TYPE "UDT_RATPositioning"
VERSION : 0.1
   STRUCT
      Lower { ExternalAccessible := 'False'; ExternalVisible := 'False'; ExternalWritable := 'False'} : Struct   // Roller part
         StartPositionA { ExternalAccessible := 'False'; ExternalVisible := 'False'; ExternalWritable := 'False'} : Int;   // Start position detected by OB30
         StartPositionB { ExternalAccessible := 'False'; ExternalVisible := 'False'; ExternalWritable := 'False'} : Int;
         EndPosition { ExternalAccessible := 'False'; ExternalVisible := 'False'; ExternalWritable := 'False'} : Int;   // End position defined by RAT FB
         Start { ExternalAccessible := 'False'; ExternalVisible := 'False'; ExternalWritable := 'False'} : Bool;   // Start command set by RAT FB
         Done { ExternalAccessible := 'False'; ExternalVisible := 'False'; ExternalWritable := 'False'} : Bool;   // MCO finish positioning
         ResetPosition { ExternalAccessible := 'False'; ExternalVisible := 'False'; ExternalWritable := 'False'} : Bool;
         PositionRequired { ExternalAccessible := 'False'; ExternalVisible := 'False'; ExternalWritable := 'False'} : Bool;
      END_STRUCT;
      Upper { ExternalAccessible := 'False'; ExternalVisible := 'False'; ExternalWritable := 'False'} : Struct   // UBT part
         StartPositionC { ExternalAccessible := 'False'; ExternalVisible := 'False'; ExternalWritable := 'False'} : Int;   // Start position detected by OB30
         StartPositionD { ExternalAccessible := 'False'; ExternalVisible := 'False'; ExternalWritable := 'False'} : Int;
         EndPosition { ExternalAccessible := 'False'; ExternalVisible := 'False'; ExternalWritable := 'False'} : Int;   // End position defined by RAT FB
         Start { ExternalAccessible := 'False'; ExternalVisible := 'False'; ExternalWritable := 'False'} : Bool;   // Start command set by RAT FB
         Done { ExternalAccessible := 'False'; ExternalVisible := 'False'; ExternalWritable := 'False'} : Bool;   // MCO finish positioning
         ResetPosition { ExternalAccessible := 'False'; ExternalVisible := 'False'; ExternalWritable := 'False'} : Bool;
         PositionRequired { ExternalAccessible := 'False'; ExternalVisible := 'False'; ExternalWritable := 'False'} : Bool;
      END_STRUCT;
   END_STRUCT;

END_TYPE

TYPE "UDT_ValveInterface"
TITLE = UDT_ValveInterface
VERSION : 0.1
//UDT valve interface between modules
   STRUCT
      Open { ExternalAccessible := 'False'; ExternalVisible := 'False'; ExternalWritable := 'False'} : Bool;   // Interface command valve Open / Extend
      Close { ExternalAccessible := 'False'; ExternalVisible := 'False'; ExternalWritable := 'False'} : Bool;   // Interface command valve Close / Retract
      IsOpened { ExternalAccessible := 'False'; ExternalVisible := 'False'; ExternalWritable := 'False'} : Bool;   // Valve feedback opened / extended
      IsClosed { ExternalAccessible := 'False'; ExternalVisible := 'False'; ExternalWritable := 'False'} : Bool;   // Valve feedback closed / retracted
      Error { ExternalAccessible := 'False'; ExternalVisible := 'False'; ExternalWritable := 'False'} : Bool;   // Valve error
   END_STRUCT;

END_TYPE

FUNCTION "FC_Fifo" : Void
TITLE = FC_Fifo
{ S7_Optimized_Access := 'TRUE' }
AUTHOR : MHSE
FAMILY : GeneralSystemFunctions
VERSION : 3.0
// ATTRIBUTES
// AUTO_NUMBER = True
// BLOCK_NUMBER = 17
// END_ATTRIBUTES
//Function for controlling FIFO register.
   VAR_INPUT
      ic_Mode : Char;   // Mode selector: "W" - Write; "R" - Read; "C" - Clear (Reset) "S" - Status
   END_VAR

   VAR_OUTPUT
      qUDT_Status : "UDT_FifoStatus";   // FIFO status structure
      qx_Error : Bool;   // Collective error output
      qx_Warning : Bool;   // Collective warning output
   END_VAR

   VAR_IN_OUT
      iqv_Data : Variant;   // Data
      iqUDT_FifoHeader : "UDT_FifoHeader";   // FIFO header
      iqv_DataBuffer : Variant;   // FIFO data buffer
   END_VAR

   VAR_TEMP
      tUDT_Status : "UDT_FifoStatus";   // Status structure
      ti_MoveBLKErrorCode : Int;   // Move_BLK_Variant function return
      tx_HeaderValid : Bool;   // Header valid
   END_VAR


BEGIN
	(*
	----------------------------------------------------------------------------------------

	Version history:
	Date        | Version   | Author        | Remark
	----------------------------------------------------------------------------------------
	24/05/2019  | 0.1       | L.Klar        | first release MHS TIA 15.1
	14/06/2019  | 0.2       | A.Nowak       | Replacement of instruction if for direct write into variable - Region 3 , 4.1 , 4.2 , 4.3 , 4.4 , 8.1  , 8.2
	17/07/2019  | 0.3       | L.Klar        | Status handling changed
	24/07/2019  | 2.0       | L.Klar        | 2.0 MHS library release TIA 15.1
	23/08/2019  | 2.1       | K.Pokorski    | Comments corrected
	27/08/2019  | 2.2       | M.Kurpiers    | Comments adjusted
	27/09/2019  | 2.3       | K.Pokorski    | Variant input included
	01/10/2019  | 2.4       | A.Nowak       | Correct comments and rename regions
	12/11/2019  | 3.0       | P.Majka       | 3.0 MHS library release TIA 15.1
	21/02/2023  | 4.0       | F.Baten       | 4.0 Release TIA 17.5
	*)

	REGION 1 – Diagnostic bits initialization

	    // Clear FIFO statuses
	    #tUDT_Status.FifoFull := FALSE;
	    #tUDT_Status.FifoPreFull := FALSE;

	END_REGION

	REGION 2 – Array's information

	    // If buffer elements type is invalid, set the error
	    #tUDT_Status.InvalidDataType := NOT (TypeOf(#iqv_Data) = TypeOfElements(#iqv_DataBuffer));

	END_REGION

	REGION 3 – Mode validation

	    // Set the mode invalid if selected mode isn't one of the following: W- Write, R - Read, C - Clear, S - Status
	    #tUDT_Status.InvalidMode := #ic_Mode <> 'W'
	    AND #ic_Mode <> 'R'
	    AND #ic_Mode <> 'C'
	    AND #ic_Mode <> 'S';

	END_REGION

	REGION 4 – The header settings checking

	    // The correct mode has been selected and data type is valid
	    IF (NOT #tUDT_Status.InvalidMode
	        AND NOT #tUDT_Status.InvalidDataType)
	    THEN

	        REGION 4.1 – The number of maximum FIFO entries validation

	            // Write the number of array's elements to FIFO header
	            #iqUDT_FifoHeader.MaxNrOfEntries := "FC_GetNrOfArrayEl"(#iqv_DataBuffer);

	            // Set the invalid maximum number of entries error
	            #tUDT_Status.InvalidMaxNrOfEntries := #iqUDT_FifoHeader.MaxNrOfEntries <= 0;

	        END_REGION

	        REGION 4.2 – The number of total FIFO entries validation

	            // Set the invalid total number of entries error
	            #tUDT_Status.InvalidTotalEntriesStored := #iqUDT_FifoHeader.TotalEntriesStored < 0        // The total number of entries is lower than 0
	            OR #iqUDT_FifoHeader.TotalEntriesStored > #iqUDT_FifoHeader.MaxNrOfEntries;               // The total number of entries is greater than the maximum number of entries

	        END_REGION

	        REGION 4.3 – The number of the next entry to write

	            // Set the invalid next entry to write
	            #tUDT_Status.InvalidNextEntryToWrite := #iqUDT_FifoHeader.NextEntryToWrite < 0            // The number of next entry to write is lower than 0
	            OR #iqUDT_FifoHeader.NextEntryToWrite >= #iqUDT_FifoHeader.MaxNrOfEntries;                // The number of next entry to write is greater or equal to the maximum number of entries

	        END_REGION

	        REGION 4.4 – The number of the next entry to read

	            // Set the invalid next entry to read
	            #tUDT_Status.InvalidNextEntryToRead := #iqUDT_FifoHeader.NextEntryToRead < 0              // The number of next entry to read is lower than 0
	            OR #iqUDT_FifoHeader.NextEntryToRead >= #iqUDT_FifoHeader.MaxNrOfEntries;                 // The number of next entry to read is greater or equal to the maximum nr of entries

	        END_REGION

	        REGION 4.5 – FIFO header validation summary

	            // Create collective header error
	            #tx_HeaderValid := NOT #tUDT_Status.InvalidMaxNrOfEntries
	            AND NOT #tUDT_Status.InvalidTotalEntriesStored
	            AND NOT #tUDT_Status.InvalidNextEntryToWrite
	            AND NOT #tUDT_Status.InvalidNextEntryToRead;

	        END_REGION

	    END_IF;

	END_REGION

	REGION 5 – Writing the data into the FIFO buffer

	    IF (#ic_Mode = 'W'                                                                          // Write mode selected
	        AND #tx_HeaderValid                                                                     // FIFO header valid
	        AND NOT #tUDT_Status.InvalidDataType)                                                  // Buffer data type valid
	    THEN


	        IF (#iqUDT_FifoHeader.TotalEntriesStored < #iqUDT_FifoHeader.MaxNrOfEntries)          // Checking total number of stored entries
	        THEN

	            // Move input data to FIFO data buffer
	            #ti_MoveBLKErrorCode := MOVE_BLK_VARIANT(SRC := #iqv_Data,
	                                                     COUNT := 1,
	                                                     SRC_INDEX := 0,
	                                                     DEST_INDEX := #iqUDT_FifoHeader.NextEntryToWrite,
	                                                     DEST => #iqv_DataBuffer);

	            // Increment the number of the next entry to write
	            #iqUDT_FifoHeader.NextEntryToWrite += 1;

	            // Increment the total number of stored entries
	            #iqUDT_FifoHeader.TotalEntriesStored += 1;


	            IF (#iqUDT_FifoHeader.NextEntryToWrite >= #iqUDT_FifoHeader.MaxNrOfEntries)       // Check the number of the next entry to write
	            THEN

	                #iqUDT_FifoHeader.NextEntryToWrite := 0;

	            END_IF;

	        ELSE

	            #tUDT_Status.FifoFull := TRUE;

	        END_IF;

	    END_IF;

	END_REGION

	REGION 6 – Reading the data from the FIFO data buffer

	    IF (#ic_Mode = 'R'                                                                  // Read mode selected
	        AND #tx_HeaderValid                                                             // FIFO header valid
	        AND NOT #tUDT_Status.InvalidDataType)                                           // Buffer data type valid
	    THEN

	        IF (#iqUDT_FifoHeader.TotalEntriesStored > 0)                                   // Checking total number of stored entries
	        THEN

	            // Move the FIFO data to the data output
	            #ti_MoveBLKErrorCode := MOVE_BLK_VARIANT(SRC := #iqv_DataBuffer,
	                                                     COUNT := 1,
	                                                     SRC_INDEX := #iqUDT_FifoHeader.NextEntryToRead,
	                                                     DEST_INDEX := 0,
	                                                     DEST => #iqv_Data);

	            // Increment the number of the next entry to read
	            #iqUDT_FifoHeader.NextEntryToRead += 1;

	            // Decrement the total number of stored entries
	            #iqUDT_FifoHeader.TotalEntriesStored -= 1;

	            IF (#iqUDT_FifoHeader.NextEntryToRead >= #iqUDT_FifoHeader.MaxNrOfEntries)  // Check the number of the next entry to read
	            THEN

	                #iqUDT_FifoHeader.NextEntryToRead := 0;

	            END_IF;

	        END_IF;

	    END_IF;

	END_REGION

	REGION 7 – Clearing the FIFO header

	    IF (#ic_Mode = 'C'                      // Clear mode selected
	        AND #tx_HeaderValid)                // FIFO header valid
	    THEN

	        #iqUDT_FifoHeader.TotalEntriesStored := 0;
	        #iqUDT_FifoHeader.NextEntryToWrite := 0;
	        #iqUDT_FifoHeader.NextEntryToRead := 0;

	    END_IF;

	END_REGION

	REGION 8 – FIFO management status update

	    IF (#tx_HeaderValid)                   // The header is valid
	    THEN

	        REGION 8.1 – FIFO Empty

	            // Set the FIFO empty status bit
	            #iqUDT_FifoHeader.Status.Empty := #iqUDT_FifoHeader.TotalEntriesStored = 0;

	        END_REGION

	        REGION 8.2 – FIFO Full

	            // Set the FIFO full status bit
	            #iqUDT_FifoHeader.Status.Full := #iqUDT_FifoHeader.TotalEntriesStored = #iqUDT_FifoHeader.MaxNrOfEntries;

	        END_REGION

	        REGION 8.3 – FIFO Pre-full

	            IF (#iqUDT_FifoHeader.TotalEntriesStored >= 0.9 * #iqUDT_FifoHeader.MaxNrOfEntries)       // Checking if the number of total stored entries is greater or equal to 90% of the max number of entries
	            THEN

	                // Set the FIFO pre-full status
	                #iqUDT_FifoHeader.Status.Prefull := TRUE;
	                #tUDT_Status.FifoPreFull := TRUE;

	            ELSE

	                #iqUDT_FifoHeader.Status.Prefull := FALSE;

	            END_IF;

	        END_REGION

	    END_IF;

	END_REGION

	REGION 9 – Status

	    REGION 9.1 – Common status update

	        // Collective error output
	        #qx_Error := NOT #tx_HeaderValid
	        OR #tUDT_Status.InvalidMode
	        OR #tUDT_Status.FifoFull
	        OR #tUDT_Status.InvalidDataType;

	        // Collective warning output
	        #qx_Warning := #tUDT_Status.FifoPreFull;

	    END_REGION

	    REGION 9.2 – Status update

	        // Update the outer status structure with internal status structure
	        #qUDT_Status := #tUDT_Status;

	    END_REGION

	END_REGION
END_FUNCTION

TYPE "UDT_VfdNordPI"
TITLE = UDT_VfdNordPI
VERSION : 0.1
//User-defined structure of VFD Nord input telegram.
   STRUCT
      ZSW : Struct   // Status word
         SetpointReached { ExternalAccessible := 'False'; ExternalVisible := 'False'; ExternalWritable := 'False'} : Bool;   // 0 = Actual value does not corresponf to setpoint. 1 = Actual value matches the setpoint
         BusControlActive { ExternalAccessible := 'False'; ExternalVisible := 'False'; ExternalWritable := 'False'} : Bool;   // 0 = Control on local device active. 1 = The master has beed requestd to take over control
         "StartFunction481.9" { ExternalAccessible := 'False'; ExternalVisible := 'False'; ExternalWritable := 'False'} : Bool;   // 1 = Bus bit 10 of status word is set P481
         RotationRightIsOn { ExternalAccessible := 'False'; ExternalVisible := 'False'; ExternalWritable := 'False'} : Bool;   // 1 = The FI output voltage has a RH rotation field
         RotationLeftIsOn { ExternalAccessible := 'False'; ExternalVisible := 'False'; ExternalWritable := 'False'} : Bool;   // 1 = The FI output voltage has a LH rotation field
         "StartFunction481.10" { ExternalAccessible := 'False'; ExternalVisible := 'False'; ExternalWritable := 'False'} : Bool;   // 1 = Bus bit 13 of status word is set P481
         ParameterSetBit0ON { ExternalAccessible := 'False'; ExternalVisible := 'False'; ExternalWritable := 'False'} : Bool;   // Parameter set bit 0 status
         ParameterSetBit1ON { ExternalAccessible := 'False'; ExternalVisible := 'False'; ExternalWritable := 'False'} : Bool;   // Parameter set bit 0 status
         ReadyToStart { ExternalAccessible := 'False'; ExternalVisible := 'False'; ExternalWritable := 'False'} : Bool;   // 1 = Initialisation completed, charging relay switched on, output voltage disabled
         ReadyForOperation { ExternalAccessible := 'False'; ExternalVisible := 'False'; ExternalWritable := 'False'} : Bool;   // 0 = No switch-on command present or fault. 1 = The inverted can start with the command "Enable operation"
         OperationEnabled { ExternalAccessible := 'False'; ExternalVisible := 'False'; ExternalWritable := 'False'} : Bool;   // 1 = The output voltage is enabled; ramp of the frequency inverter up to the existing setpoint
         Fault : Bool := FALSE;   // 1 = Drive unit defective, not ready for operation
         VoltageEnabled { ExternalAccessible := 'False'; ExternalVisible := 'False'; ExternalWritable := 'False'} : Bool;   // 0 = "Disable voltage" command present
         EmergencyStop { ExternalAccessible := 'False'; ExternalVisible := 'False'; ExternalWritable := 'False'} : Bool;   // 0 = "Emergency stop" command present
         StartingDisabled { ExternalAccessible := 'False'; ExternalVisible := 'False'; ExternalWritable := 'False'} : Bool;   // 1 = With the command "Standby" the FI goes into status "Ready to switch on"
         WarningActive { ExternalAccessible := 'False'; ExternalVisible := 'False'; ExternalWritable := 'False'} : Bool;   // 1 = Drive operation continues, no acknowledgement necessary
      END_STRUCT;
      ActualSpeed : Int;   // Actual calculated speed [rpm]. [Range  -200% ..200%][100%=4000HEX/ 16384DEC = P202 nominal speed]
      FaultCode : Int;   // Actual fault code
   END_STRUCT;

END_TYPE

DATA_BLOCK "DB_GINDefault"
{ S7_Optimized_Access := 'TRUE' }
VERSION : 0.1
NON_RETAIN
   VAR
      GIN { ExternalAccessible := 'False'; ExternalVisible := 'False'; ExternalWritable := 'False'; S7_SetPoint := 'False'} : Array[1..20] of "UDT_GIN";   // GIN informations
   END_VAR


BEGIN

END_DATA_BLOCK

FUNCTION_BLOCK "FB_VfdNORDCommissioning"
TITLE = Block for parameterising NORD VFD
{ S7_Optimized_Access := 'TRUE' }
VERSION : 0.1
// ATTRIBUTES
// AUTO_NUMBER = True
// BLOCK_NUMBER = 234
// END_ATTRIBUTES
   VAR_INPUT
      ihw_HardwareID { ExternalAccessible := 'False'; ExternalVisible := 'False'; ExternalWritable := 'False'} : HW_IO := 0;   // Device hardware ID
      iudt_MotorData { ExternalAccessible := 'False'; ExternalVisible := 'False'; ExternalWritable := 'False'} : "UDT_MotorData";
      ir_ReferenceFrequency { ExternalAccessible := 'False'; ExternalVisible := 'False'; ExternalWritable := 'False'} : Real;
      ix_VFDReadyToRun { ExternalAccessible := 'False'; ExternalVisible := 'False'; ExternalWritable := 'False'} : Bool;   // Condition to start motor identyfication
   END_VAR

   VAR_OUTPUT
      qi_HWAdress { ExternalAccessible := 'False'; ExternalVisible := 'False'; ExternalWritable := 'False'} : Int;
      qx_Busy { ExternalAccessible := 'False'; ExternalVisible := 'False'; ExternalWritable := 'False'} : Bool;   // Parametrisation in progress
      qx_Done { ExternalAccessible := 'False'; ExternalVisible := 'False'; ExternalWritable := 'False'} : Bool;   // Parametrisation done
      qx_Error { ExternalAccessible := 'False'; ExternalVisible := 'False'; ExternalWritable := 'False'} : Bool;   // Parametrisation error
      qx_24VCommissioningDone { ExternalAccessible := 'False'; ExternalVisible := 'False'; ExternalWritable := 'False'} : Bool;   // 24V commissioning done succesfully
   END_VAR

   VAR_IN_OUT
      iqx_Enable { ExternalAccessible := 'False'; ExternalVisible := 'False'; ExternalWritable := 'False'} : Bool;   // Input enable signal
   END_VAR

   VAR
      sFB_ParaAcycRead { ExternalAccessible := 'False'; ExternalVisible := 'False'; ExternalWritable := 'False'; S7_SetPoint := 'False'} : "FB_VfdNORDParaAcycRead";
      sFB_ParaAcycWrite { ExternalAccessible := 'False'; ExternalVisible := 'False'; ExternalWritable := 'False'; S7_SetPoint := 'False'} : "FB_VfdNORDParaAcycWrite";
      sR_TRIG_Done {InstructionName := 'R_TRIG'; LibVersion := '1.0'; ExternalAccessible := 'False'; ExternalVisible := 'False'; ExternalWritable := 'False'; S7_SetPoint := 'False'} : R_TRIG;
      sR_TRIG_StartJob {InstructionName := 'R_TRIG'; LibVersion := '1.0'; ExternalAccessible := 'False'; ExternalVisible := 'False'; ExternalWritable := 'False'; S7_SetPoint := 'False'} : R_TRIG;   // Bit for start trigger for rising edge
      sF_TRIG_CancelJob {InstructionName := 'F_TRIG'; LibVersion := '1.0'; ExternalAccessible := 'False'; ExternalVisible := 'False'; ExternalWritable := 'False'; S7_SetPoint := 'False'} : F_TRIG;   // Bit for start trigger for falling edge
      sa_Parameter { ExternalAccessible := 'False'; ExternalVisible := 'False'; ExternalWritable := 'False'; S7_SetPoint := 'False'} : Array[0..60] of "UDT_VfdNordParameter";   // Data of parameters
      sa_Status { ExternalAccessible := 'False'; ExternalVisible := 'False'; ExternalWritable := 'False'} : Struct   // Parametrization status
         StepNrError { ExternalAccessible := 'False'; ExternalVisible := 'False'; ExternalWritable := 'False'} : Int;   // The number of the step in witch the error occurred
         ParameterNrError { ExternalAccessible := 'False'; ExternalVisible := 'False'; ExternalWritable := 'False'} : Int;   // The number of the parameter in witch the error occurred
         StepNr { ExternalAccessible := 'False'; ExternalVisible := 'False'; ExternalWritable := 'False'} : Int := 0;   // Current step number
         ResponseValueError { ExternalAccessible := 'False'; ExternalVisible := 'False'; ExternalWritable := 'False'} : Bool;   // Response value error
         WrongFormat { ExternalAccessible := 'False'; ExternalVisible := 'False'; ExternalWritable := 'False'} : Bool;   // Wrong parameter format
         TimeExceeded { ExternalAccessible := 'False'; ExternalVisible := 'False'; ExternalWritable := 'False'} : Bool;   // Time has been exceeded
         NeedAck { ExternalAccessible := 'False'; ExternalVisible := 'False'; ExternalWritable := 'False'} : Bool;   // Need acknowledge signal (to cintinue parametrization)
         StepDone { ExternalAccessible := 'False'; ExternalVisible := 'False'; ExternalWritable := 'False'} : Bool;   // Step done
      END_STRUCT;
      si_StepTime { ExternalAccessible := 'False'; ExternalVisible := 'False'; ExternalWritable := 'False'} : Int;
      si_StepMax { ExternalAccessible := 'False'; ExternalVisible := 'False'; ExternalWritable := 'False'} : Int := 0;   // Maximum step number
      sx_Start { ExternalAccessible := 'False'; ExternalVisible := 'False'; ExternalWritable := 'False'} : Bool;   // Signal to start of parameterization function SinaPara
      sx_Busy { ExternalAccessible := 'False'; ExternalVisible := 'False'; ExternalWritable := 'False'} : Bool;   // Parametrization in progress (busy)
      sx_Done { ExternalAccessible := 'False'; ExternalVisible := 'False'; ExternalWritable := 'False'} : Bool;   // Parametrization done
      sx_Error { ExternalAccessible := 'False'; ExternalVisible := 'False'; ExternalWritable := 'False'} : Bool;   // Main error signal
      sx_PreparedData { ExternalAccessible := 'False'; ExternalVisible := 'False'; ExternalWritable := 'False'} : Bool;   // Step data prepared
      sx_ReadOrder { ExternalAccessible := 'False'; ExternalVisible := 'False'; ExternalWritable := 'False'} : Bool;   // Order to read paraeter with transition from 0 to 1
      sx_WriteOrder { ExternalAccessible := 'False'; ExternalVisible := 'False'; ExternalWritable := 'False'} : Bool;   // Order to write parameter with transition from 0 to 1
      sx_MaxStepCalculation { ExternalAccessible := 'False'; ExternalVisible := 'False'; ExternalWritable := 'False'} : Bool;   // Maximum step calculated
   END_VAR
   VAR RETAIN
      sx_24VCommissioningDone { ExternalAccessible := 'False'; ExternalVisible := 'False'; ExternalWritable := 'False'} : Bool;   // 24V commissioning done succesfully
   END_VAR

   VAR_TEMP
      ti_index : Int;   // Temporary array index
      ti_ControlMethod : Int;
      ti_EncoderCode : Int;
      ti_i : Int;   // Loop counter
      ti_BrakeReaction : Int;
   END_VAR

   VAR CONSTANT
      ci_CFC_ClosedLoop : Int := 1;
      ci_CFC_OpenLoop : Int := 0;
      ci_EncoderRes512 : Int := 1;
      ci_EncoderRes1024 : Int := 3;
      ci_EncoderRes2048 : Int := 5;
      ci_EncoderRes4096 : Int := 6;
      ci_MaxStepTime : Int := 100;
   END_VAR


BEGIN
	(*
	----------------------------------------------------------------------------------------

	Version history:
	Date        | Version   | Author        | Remark
	----------------------------------------------------------------------------------------
	12/01/2020  | 0.1       | S.Theocharis  | Initial version TIA 15.1
	08/04/2021  | 0.2       | F.Baten       | New read/write blocks
	                                        | New motor parameter set ( most values not 32bit )
	                                        | PN device with onboard safety
	                                        | Reading and writing optimised
	27/01/2022  | 0.3       | K.Pokorski    | Add 24V and 400V commissionig status
	                                        | Fix VFD Output bug
	                                        | Initialize InUse status in all parameters
	                                        | Fix Motor identification
	                                        | Save parameters to External memory
	                                        | Delete saving F-parameters from sequence (not working and creating faults)
	                                        | Delete reading CRC code (reading old CRC code what can be confusing)
	21/04/2022  | 0.4       | K.Pokorski    | Delete motor identification
	21/02/2023  | 4.0       | F.Baten       | 4.0 Release TIA 17.5

	*)

	REGION 1 - Start Job

	    // Monitor rising trigger if is input enable signal
	    #sR_TRIG_StartJob(CLK := #iqx_Enable);

	    IF (#sR_TRIG_StartJob.Q)
	    THEN
	        #sx_Start := TRUE;
	        #sx_Busy := TRUE;
	        #sx_Done := FALSE;
	        #sx_Error := FALSE;
	        #sx_PreparedData := FALSE;
	        #sx_MaxStepCalculation := FALSE;
	        #sa_Status.StepDone := FALSE;
	        #sa_Status.StepNrError := 0;
	        #sa_Status.ParameterNrError := 0;
	        #sa_Status.StepNr := 0;
	        #si_StepTime := 0;
	        #qi_HWAdress := 0;

	        FOR #ti_i := 0 TO 60 DO
	            #sa_Parameter[#ti_i].InUse := FALSE;
	        END_FOR;



	    END_IF;

	END_REGION

	REGION 2 - Build Sequences in static memory

	    IF #sR_TRIG_StartJob.Q THEN
	        //  IF NOT #sx_24VCommissioningDone THEN
	        REGION Step 01 - P523 Factory reset [0..3]
	            #ti_index := 0;
	            #sa_Parameter[#ti_index].ParaNumber := 523;
	            #sa_Parameter[#ti_index].Index := 0;
	            #sa_Parameter[#ti_index].WriteValue := 1;
	            #sa_Parameter[#ti_index].WriteAccess := TRUE;
	            #sa_Parameter[#ti_index].ParaSet := 0;
	            #sa_Parameter[#ti_index].Format32 := FALSE;
	            #sa_Parameter[#ti_index].ActualValue := 0;
	            #sa_Parameter[#ti_index].InUse := TRUE;
	            #sa_Parameter[#ti_index].RamOnly := FALSE;
	        END_REGION

	        REGION Step 02 - P003 Set supervisor code to access all parameters [0..9999]
	            #ti_index := #ti_index + 1;
	            #sa_Parameter[#ti_index].ParaNumber := 3;
	            #sa_Parameter[#ti_index].Index := 0;
	            #sa_Parameter[#ti_index].WriteValue := 3;
	            #sa_Parameter[#ti_index].WriteAccess := TRUE;
	            #sa_Parameter[#ti_index].ParaSet := 0;
	            #sa_Parameter[#ti_index].Format32 := FALSE;
	            #sa_Parameter[#ti_index].ActualValue := 0;
	            #sa_Parameter[#ti_index].InUse := TRUE;
	            #sa_Parameter[#ti_index].RamOnly := FALSE;
	        END_REGION

	        REGION Step 03 - P800 Set Operating mode Safety [0-1]
	            #ti_index := #ti_index + 1;
	            #sa_Parameter[#ti_index].ParaNumber := 800;
	            #sa_Parameter[#ti_index].Index := 1;
	            #sa_Parameter[#ti_index].WriteValue := 1;
	            #sa_Parameter[#ti_index].WriteAccess := TRUE;
	            #sa_Parameter[#ti_index].ParaSet := 0;
	            #sa_Parameter[#ti_index].Format32 := FALSE;
	            #sa_Parameter[#ti_index].ActualValue := 0;
	            #sa_Parameter[#ti_index].InUse := TRUE;
	            #sa_Parameter[#ti_index].RamOnly := FALSE;
	        END_REGION

	        REGION Step 04 - P800 Set Operating mode Safety [0-1]
	            #ti_index := #ti_index + 1;
	            #sa_Parameter[#ti_index].ParaNumber := 800;
	            #sa_Parameter[#ti_index].Index := 2;
	            #sa_Parameter[#ti_index].WriteValue := 0;
	            #sa_Parameter[#ti_index].WriteAccess := TRUE;
	            #sa_Parameter[#ti_index].ParaSet := 0;
	            #sa_Parameter[#ti_index].Format32 := FALSE;
	            #sa_Parameter[#ti_index].ActualValue := 0;
	            #sa_Parameter[#ti_index].InUse := TRUE;
	            #sa_Parameter[#ti_index].RamOnly := FALSE;
	        END_REGION

	        REGION Step 05 - P802 Set Enable safety channel [0-1]  Channel 1 on
	            #ti_index := #ti_index + 1;
	            #sa_Parameter[#ti_index].ParaNumber := 802;
	            #sa_Parameter[#ti_index].Index := 1;
	            #sa_Parameter[#ti_index].WriteValue := 1;
	            #sa_Parameter[#ti_index].WriteAccess := TRUE;
	            #sa_Parameter[#ti_index].ParaSet := 0;
	            #sa_Parameter[#ti_index].Format32 := FALSE;
	            #sa_Parameter[#ti_index].ActualValue := 0;
	            #sa_Parameter[#ti_index].InUse := TRUE;
	            #sa_Parameter[#ti_index].RamOnly := FALSE;
	        END_REGION

	        REGION Step 06 - P802 Set Enable safety channel [0-1]  Channel 2 on
	            #ti_index := #ti_index + 1;
	            #sa_Parameter[#ti_index].ParaNumber := 802;
	            #sa_Parameter[#ti_index].Index := 2;
	            #sa_Parameter[#ti_index].WriteValue := 1;
	            #sa_Parameter[#ti_index].WriteAccess := TRUE;
	            #sa_Parameter[#ti_index].ParaSet := 0;
	            #sa_Parameter[#ti_index].Format32 := FALSE;
	            #sa_Parameter[#ti_index].ActualValue := 0;
	            #sa_Parameter[#ti_index].InUse := TRUE;
	            #sa_Parameter[#ti_index].RamOnly := FALSE;
	        END_REGION

	        REGION Step 07 - P802 Set Enable safety channel [0-1]  Channel 3 on
	            #ti_index := #ti_index + 1;
	            #sa_Parameter[#ti_index].ParaNumber := 802;
	            #sa_Parameter[#ti_index].Index := 3;
	            #sa_Parameter[#ti_index].WriteValue := 1;
	            #sa_Parameter[#ti_index].WriteAccess := TRUE;
	            #sa_Parameter[#ti_index].ParaSet := 0;
	            #sa_Parameter[#ti_index].Format32 := FALSE;
	            #sa_Parameter[#ti_index].ActualValue := 0;
	            #sa_Parameter[#ti_index].InUse := TRUE;
	            #sa_Parameter[#ti_index].RamOnly := FALSE;
	        END_REGION

	        REGION Step 08 - P846 Read dipswitches
	            #ti_index := #ti_index + 1;
	            #sa_Parameter[#ti_index].ParaNumber := 846;
	            #sa_Parameter[#ti_index].Index := 0;
	            #sa_Parameter[#ti_index].WriteValue := 0;
	            #sa_Parameter[#ti_index].WriteAccess := FALSE;
	            #sa_Parameter[#ti_index].ParaSet := 0;
	            #sa_Parameter[#ti_index].Format32 := FALSE;
	            #sa_Parameter[#ti_index].ActualValue := 0;
	            #sa_Parameter[#ti_index].InUse := TRUE;
	            #sa_Parameter[#ti_index].RamOnly := FALSE;
	        END_REGION

	        REGION Step 09 - P120 Set extern control units [0-1]  Switch off 3 and 4
	            #ti_index := #ti_index + 1;
	            #sa_Parameter[#ti_index].ParaNumber := 120;
	            #sa_Parameter[#ti_index].Index := 3;
	            #sa_Parameter[#ti_index].WriteValue := 0;
	            #sa_Parameter[#ti_index].WriteAccess := TRUE;
	            #sa_Parameter[#ti_index].ParaSet := 0;
	            #sa_Parameter[#ti_index].Format32 := FALSE;
	            #sa_Parameter[#ti_index].ActualValue := 0;
	            #sa_Parameter[#ti_index].InUse := TRUE;
	            #sa_Parameter[#ti_index].RamOnly := FALSE;
	        END_REGION

	        REGION Step 10 - P120 Set extern control units [0-1]  Switch off 3 and 4
	            #ti_index := #ti_index + 1;
	            #sa_Parameter[#ti_index].ParaNumber := 120;
	            #sa_Parameter[#ti_index].Index := 4;
	            #sa_Parameter[#ti_index].WriteValue := 0;
	            #sa_Parameter[#ti_index].WriteAccess := TRUE;
	            #sa_Parameter[#ti_index].ParaSet := 0;
	            #sa_Parameter[#ti_index].Format32 := FALSE;
	            #sa_Parameter[#ti_index].ActualValue := 0;
	            #sa_Parameter[#ti_index].InUse := TRUE;
	            #sa_Parameter[#ti_index].RamOnly := FALSE;
	        END_REGION

	        REGION Step 11 - P202 Write motor nominal speed [150...24000]rpm
	            #ti_index := #ti_index + 1;
	            #sa_Parameter[#ti_index].ParaNumber := 202;
	            #sa_Parameter[#ti_index].Index := 0;
	            #sa_Parameter[#ti_index].WriteValue := #iudt_MotorData.NominalSpeed;
	            #sa_Parameter[#ti_index].WriteAccess := TRUE;
	            #sa_Parameter[#ti_index].ParaSet := 1; // Parameter set 1
	            #sa_Parameter[#ti_index].Format32 := FALSE;
	            #sa_Parameter[#ti_index].ActualValue := 0;
	            #sa_Parameter[#ti_index].InUse := TRUE;
	            #sa_Parameter[#ti_index].RamOnly := FALSE;
	        END_REGION

	        REGION Step 12 - P203 Write motor nominal current [0.1 ...1000.0]A
	            #ti_index := #ti_index + 1;
	            #sa_Parameter[#ti_index].ParaNumber := 203;
	            #sa_Parameter[#ti_index].Index := 0;
	            #sa_Parameter[#ti_index].WriteValue := (REAL_TO_DINT(#iudt_MotorData.NominalCurrent * 10));  // Value 55 = 5.5 Amps
	            #sa_Parameter[#ti_index].WriteAccess := TRUE;
	            #sa_Parameter[#ti_index].ParaSet := 0; // Parameter set 1
	            #sa_Parameter[#ti_index].Format32 := FALSE;
	            #sa_Parameter[#ti_index].ActualValue := 0;
	            #sa_Parameter[#ti_index].InUse := TRUE;
	            #sa_Parameter[#ti_index].RamOnly := FALSE;
	        END_REGION

	        REGION Step 13 - P204 Write motor nominal voltage [100 ... 800]V
	            #ti_index := #ti_index + 1;
	            #sa_Parameter[#ti_index].ParaNumber := 204;
	            #sa_Parameter[#ti_index].Index := 0;
	            #sa_Parameter[#ti_index].WriteValue := #iudt_MotorData.NominalVoltage;
	            #sa_Parameter[#ti_index].WriteAccess := FALSE;
	            #sa_Parameter[#ti_index].ParaSet := 1; // Parameter set 1
	            #sa_Parameter[#ti_index].Format32 := FALSE;
	            #sa_Parameter[#ti_index].ActualValue := 0;
	            #sa_Parameter[#ti_index].InUse := TRUE;
	            #sa_Parameter[#ti_index].RamOnly := FALSE;
	        END_REGION

	        REGION Step 14 - P205 Write motor nominal power
	            #ti_index := #ti_index + 1;
	            #sa_Parameter[#ti_index].ParaNumber := 205;
	            #sa_Parameter[#ti_index].Index := 0;
	            #sa_Parameter[#ti_index].WriteValue := (REAL_TO_DINT(#iudt_MotorData.NominalPower * 100));
	            #sa_Parameter[#ti_index].WriteAccess := TRUE;
	            #sa_Parameter[#ti_index].ParaSet := 0; // Parameter set 1
	            #sa_Parameter[#ti_index].Format32 := FALSE;
	            #sa_Parameter[#ti_index].ActualValue := 0;
	            #sa_Parameter[#ti_index].InUse := TRUE;
	            #sa_Parameter[#ti_index].RamOnly := FALSE;
	        END_REGION

	        REGION Step 15 - P206 Write motor cosPhi [0.50 ... 0.95]
	            #ti_index := #ti_index + 1;
	            #sa_Parameter[#ti_index].ParaNumber := 206;
	            #sa_Parameter[#ti_index].Index := 0;
	            #sa_Parameter[#ti_index].WriteValue := REAL_TO_DINT(#iudt_MotorData.CosPhi * 100);
	            #sa_Parameter[#ti_index].WriteAccess := TRUE;
	            #sa_Parameter[#ti_index].ParaSet := 0; // Parameter set 1
	            #sa_Parameter[#ti_index].Format32 := FALSE;
	            #sa_Parameter[#ti_index].ActualValue := 0;
	            #sa_Parameter[#ti_index].InUse := TRUE;
	            #sa_Parameter[#ti_index].RamOnly := FALSE;
	        END_REGION

	        REGION Step 16 - P207 Connection Star / Delta [0=Star 1=Delta]
	            #ti_index := #ti_index + 1;
	            #sa_Parameter[#ti_index].ParaNumber := 207;
	            #sa_Parameter[#ti_index].Index := 0;
	            #sa_Parameter[#ti_index].WriteValue := #iudt_MotorData.Connection;
	            #sa_Parameter[#ti_index].WriteAccess := TRUE;
	            #sa_Parameter[#ti_index].ParaSet := 0; // Parameter set 1
	            #sa_Parameter[#ti_index].Format32 := FALSE;
	            #sa_Parameter[#ti_index].ActualValue := 0;
	            #sa_Parameter[#ti_index].InUse := TRUE;
	            #sa_Parameter[#ti_index].RamOnly := FALSE;
	        END_REGION

	        REGION Step 17 - P105 Write Maximum / Reference Frequency [0.1...400.0]Hz
	            #ti_index := #ti_index + 1;
	            #sa_Parameter[#ti_index].ParaNumber := 105;
	            #sa_Parameter[#ti_index].Index := 0;
	            #sa_Parameter[#ti_index].WriteValue := REAL_TO_DINT(#ir_ReferenceFrequency * 10);
	            #sa_Parameter[#ti_index].WriteAccess := TRUE;
	            #sa_Parameter[#ti_index].ParaSet := 0; // Parameter set 1
	            #sa_Parameter[#ti_index].Format32 := FALSE;
	            #sa_Parameter[#ti_index].ActualValue := 0;
	            #sa_Parameter[#ti_index].InUse := TRUE;
	            #sa_Parameter[#ti_index].RamOnly := FALSE;
	        END_REGION

	        REGION Step 18 - P107 Brake reaction
	            IF #iudt_MotorData.BrakeConfig THEN
	                #ti_BrakeReaction := 20;
	            ELSE
	                #ti_BrakeReaction := 0;
	            END_IF;

	            #ti_index := #ti_index + 1;
	            #sa_Parameter[#ti_index].ParaNumber := 107;
	            #sa_Parameter[#ti_index].Index := 0;
	            #sa_Parameter[#ti_index].WriteValue := #ti_BrakeReaction;
	            #sa_Parameter[#ti_index].WriteAccess := TRUE;
	            #sa_Parameter[#ti_index].ParaSet := 0; // Parameter set 1
	            #sa_Parameter[#ti_index].Format32 := FALSE;
	            #sa_Parameter[#ti_index].ActualValue := 0;
	            #sa_Parameter[#ti_index].InUse := TRUE;
	            #sa_Parameter[#ti_index].RamOnly := FALSE;
	        END_REGION

	        REGION Step 19 - P300 Mode [0..2]
	            //If an IE4 motor is operated in CFC closed loop mode , the slip error monitoring must be activated. P327<>0
	            IF #iudt_MotorData.EncoderResolution <> 0 THEN
	                #ti_ControlMethod := #ci_CFC_ClosedLoop; //CFC closed loop control. Speed control with encoder feedback
	            ELSE
	                #ti_ControlMethod := #ci_CFC_OpenLoop; //VFC open loop control. Speed control without encoder feedback
	            END_IF;
	            #ti_index := #ti_index + 1;
	            #sa_Parameter[#ti_index].ParaNumber := 300;
	            #sa_Parameter[#ti_index].Index := 0;
	            #sa_Parameter[#ti_index].WriteValue := #ti_ControlMethod;
	            #sa_Parameter[#ti_index].WriteAccess := TRUE;
	            #sa_Parameter[#ti_index].ParaSet := 1; // Parameter set 1
	            #sa_Parameter[#ti_index].Format32 := FALSE;
	            #sa_Parameter[#ti_index].ActualValue := 0;
	            #sa_Parameter[#ti_index].InUse := TRUE;
	            #sa_Parameter[#ti_index].RamOnly := FALSE;
	        END_REGION

	        REGION Step 20 - P301 Encoder Resolution [0..17]
	            CASE #iudt_MotorData.EncoderResolution OF
	                512:
	                    #ti_EncoderCode := #ci_EncoderRes512;
	                1024:
	                    #ti_EncoderCode := #ci_EncoderRes1024;
	                2048:
	                    #ti_EncoderCode := #ci_EncoderRes2048;
	                4096:
	                    #ti_EncoderCode := #ci_EncoderRes4096;
	                ELSE
	                    #ti_EncoderCode := 6; //default value
	            END_CASE;

	            #ti_index := #ti_index + 1;
	            #sa_Parameter[#ti_index].ParaNumber := 301;
	            #sa_Parameter[#ti_index].Index := 0;
	            #sa_Parameter[#ti_index].WriteValue := #ti_EncoderCode;
	            #sa_Parameter[#ti_index].WriteAccess := TRUE;
	            #sa_Parameter[#ti_index].ParaSet := 0;
	            #sa_Parameter[#ti_index].Format32 := FALSE;
	            #sa_Parameter[#ti_index].ActualValue := 0;
	            #sa_Parameter[#ti_index].InUse := TRUE;
	            #sa_Parameter[#ti_index].RamOnly := FALSE;
	        END_REGION

	        REGION Step 21 - P326 Encoder ratio [0.01 ... 100.0]
	            #ti_index := #ti_index + 1;
	            #sa_Parameter[#ti_index].ParaNumber := 326;
	            #sa_Parameter[#ti_index].Index := 0;
	            #sa_Parameter[#ti_index].WriteValue := (1 * 100); //leave temporary the default 1.00;
	            #sa_Parameter[#ti_index].WriteAccess := TRUE;
	            #sa_Parameter[#ti_index].ParaSet := 0;
	            #sa_Parameter[#ti_index].Format32 := FALSE;
	            #sa_Parameter[#ti_index].ActualValue := 0;
	            #sa_Parameter[#ti_index].InUse := TRUE;
	            #sa_Parameter[#ti_index].RamOnly := FALSE;
	        END_REGION

	        REGION Step 22 - P420[1] Digital inputs [0 ... 80] DI1
	            #ti_index := #ti_index + 1;
	            #sa_Parameter[#ti_index].ParaNumber := 420;
	            #sa_Parameter[#ti_index].Index := 1;
	            #sa_Parameter[#ti_index].WriteValue := 0;
	            #sa_Parameter[#ti_index].WriteAccess := TRUE;
	            #sa_Parameter[#ti_index].ParaSet := 0;
	            #sa_Parameter[#ti_index].Format32 := FALSE;
	            #sa_Parameter[#ti_index].ActualValue := 0;
	            #sa_Parameter[#ti_index].InUse := TRUE;
	            #sa_Parameter[#ti_index].RamOnly := FALSE;
	        END_REGION

	        REGION Step 23 - P420[2] Digital inputs [0 ... 80] DI2
	            #ti_index := #ti_index + 1;
	            #sa_Parameter[#ti_index].ParaNumber := 420;
	            #sa_Parameter[#ti_index].Index := 2;
	            #sa_Parameter[#ti_index].WriteValue := 0;
	            #sa_Parameter[#ti_index].WriteAccess := TRUE;
	            #sa_Parameter[#ti_index].ParaSet := 0;
	            #sa_Parameter[#ti_index].Format32 := FALSE;
	            #sa_Parameter[#ti_index].ActualValue := 0;
	            #sa_Parameter[#ti_index].InUse := TRUE;
	            #sa_Parameter[#ti_index].RamOnly := FALSE;
	        END_REGION

	        REGION Step 24 - P420[3] Digital inputs [0 ... 80] DI3
	            #ti_index := #ti_index + 1;
	            #sa_Parameter[#ti_index].ParaNumber := 420;
	            #sa_Parameter[#ti_index].Index := 3;
	            #sa_Parameter[#ti_index].WriteValue := 0;
	            #sa_Parameter[#ti_index].WriteAccess := TRUE;
	            #sa_Parameter[#ti_index].ParaSet := 0;
	            #sa_Parameter[#ti_index].Format32 := FALSE;
	            #sa_Parameter[#ti_index].ActualValue := 0;
	            #sa_Parameter[#ti_index].InUse := TRUE;
	            #sa_Parameter[#ti_index].RamOnly := FALSE;
	        END_REGION

	        REGION Step 25 - P426 Quick Stop time [0 ... 320.00] sec
	            #ti_index := #ti_index + 1;
	            #sa_Parameter[#ti_index].ParaNumber := 426;
	            #sa_Parameter[#ti_index].Index := 0;
	            #sa_Parameter[#ti_index].WriteValue := 60;
	            #sa_Parameter[#ti_index].WriteAccess := TRUE;
	            #sa_Parameter[#ti_index].ParaSet := 1; //paraset 1
	            #sa_Parameter[#ti_index].Format32 := FALSE;
	            #sa_Parameter[#ti_index].ActualValue := 0;
	            #sa_Parameter[#ti_index].InUse := TRUE;
	            #sa_Parameter[#ti_index].RamOnly := FALSE;
	        END_REGION

	        REGION Step 26 - P509 Control word source [0..4]
	            #ti_index := #ti_index + 1;
	            #sa_Parameter[#ti_index].ParaNumber := 509;
	            #sa_Parameter[#ti_index].Index := 0;
	            #sa_Parameter[#ti_index].WriteValue := 3; // System bus communication (PN)
	            #sa_Parameter[#ti_index].WriteAccess := TRUE;
	            #sa_Parameter[#ti_index].ParaSet := 0;
	            #sa_Parameter[#ti_index].Format32 := FALSE;
	            #sa_Parameter[#ti_index].ActualValue := 0;
	            #sa_Parameter[#ti_index].InUse := TRUE;
	            #sa_Parameter[#ti_index].RamOnly := FALSE;
	        END_REGION

	        REGION Step 27 - P543[1] Actual speed to actual value 1 [0..57]
	            #ti_index := #ti_index + 1;
	            #sa_Parameter[#ti_index].ParaNumber := 543;
	            #sa_Parameter[#ti_index].Index := 1;
	            #sa_Parameter[#ti_index].WriteValue := 1; // 2 = Set Actual value 1 to actual speed
	            #sa_Parameter[#ti_index].WriteAccess := TRUE;
	            #sa_Parameter[#ti_index].ParaSet := 1; // Parameter set 1
	            #sa_Parameter[#ti_index].Format32 := FALSE;
	            #sa_Parameter[#ti_index].ActualValue := 0;
	            #sa_Parameter[#ti_index].InUse := TRUE;
	            #sa_Parameter[#ti_index].RamOnly := FALSE;
	        END_REGION

	        REGION Step 28 - P543[2] Error code to actual value 2 [0..57]
	            #ti_index := #ti_index + 1;
	            #sa_Parameter[#ti_index].ParaNumber := 543;
	            #sa_Parameter[#ti_index].Index := 2;
	            #sa_Parameter[#ti_index].WriteValue := 9; // 9 =  Set Actual value 2 to error code
	            #sa_Parameter[#ti_index].WriteAccess := TRUE;
	            #sa_Parameter[#ti_index].ParaSet := 1; // Parameter set 1
	            #sa_Parameter[#ti_index].Format32 := FALSE;
	            #sa_Parameter[#ti_index].ActualValue := 0;
	            #sa_Parameter[#ti_index].InUse := TRUE;
	            #sa_Parameter[#ti_index].RamOnly := FALSE;
	        END_REGION

	        REGION Step 29 - P543[3] DIO status to actual value 3 [0..57]
	            #ti_index := #ti_index + 1;
	            #sa_Parameter[#ti_index].ParaNumber := 543;
	            #sa_Parameter[#ti_index].Index := 3;
	            #sa_Parameter[#ti_index].WriteValue := 5; // 5 =  Set Actual value 3 to DIO status
	            #sa_Parameter[#ti_index].WriteAccess := TRUE;
	            #sa_Parameter[#ti_index].ParaSet := 1; // Parameter set 1
	            #sa_Parameter[#ti_index].Format32 := FALSE;
	            #sa_Parameter[#ti_index].ActualValue := 0;
	            #sa_Parameter[#ti_index].InUse := TRUE;
	            #sa_Parameter[#ti_index].RamOnly := FALSE;
	        END_REGION

	        REGION Step 30 - P546[1] Frequency setpoint to setpoint 1 [0..36]
	            #ti_index := #ti_index + 1;
	            #sa_Parameter[#ti_index].ParaNumber := 546;
	            #sa_Parameter[#ti_index].Index := 1;
	            #sa_Parameter[#ti_index].WriteValue := 1; // 5 =  Set setpoint 1 to frequency setpoint
	            #sa_Parameter[#ti_index].WriteAccess := TRUE;
	            #sa_Parameter[#ti_index].ParaSet := 1; // Parameter set 1
	            #sa_Parameter[#ti_index].Format32 := FALSE;
	            #sa_Parameter[#ti_index].ActualValue := 0;
	            #sa_Parameter[#ti_index].InUse := TRUE;
	            #sa_Parameter[#ti_index].RamOnly := FALSE;
	        END_REGION

	        REGION Step 31 - P546[2] Ramp setpoint to setpoint 2 [0..36]
	            #ti_index := #ti_index + 1;
	            #sa_Parameter[#ti_index].ParaNumber := 546;
	            #sa_Parameter[#ti_index].Index := 2;
	            #sa_Parameter[#ti_index].WriteValue := 15; // 15 =  Set setpoint 2 to ramp setpoint
	            #sa_Parameter[#ti_index].WriteAccess := TRUE;
	            #sa_Parameter[#ti_index].ParaSet := 1; // Parameter set 1
	            #sa_Parameter[#ti_index].Format32 := FALSE;
	            #sa_Parameter[#ti_index].ActualValue := 0;
	            #sa_Parameter[#ti_index].InUse := TRUE;
	            #sa_Parameter[#ti_index].RamOnly := FALSE;
	        END_REGION

	        REGION Step 32 - P546[3] DO control to setpoint 3 [0..36]
	            #ti_index := #ti_index + 1;
	            #sa_Parameter[#ti_index].ParaNumber := 546;
	            #sa_Parameter[#ti_index].Index := 3;
	            #sa_Parameter[#ti_index].WriteValue := 31; // 5 =  Set setpoint 3 to DIO
	            #sa_Parameter[#ti_index].WriteAccess := TRUE;
	            #sa_Parameter[#ti_index].ParaSet := 1; // Parameter set 1
	            #sa_Parameter[#ti_index].Format32 := FALSE;
	            #sa_Parameter[#ti_index].ActualValue := 0;
	            #sa_Parameter[#ti_index].InUse := TRUE;
	            #sa_Parameter[#ti_index].RamOnly := FALSE;
	        END_REGION

	        REGION Step 33 - P434[3] DO Function [1..2]
	            #ti_index := #ti_index + 1;
	            #sa_Parameter[#ti_index].ParaNumber := 434;
	            #sa_Parameter[#ti_index].Index := 1;
	            #sa_Parameter[#ti_index].WriteValue := 38;
	            #sa_Parameter[#ti_index].WriteAccess := TRUE;
	            #sa_Parameter[#ti_index].ParaSet := 1; // Parameter set 1
	            #sa_Parameter[#ti_index].Format32 := FALSE;
	            #sa_Parameter[#ti_index].ActualValue := 0;
	            #sa_Parameter[#ti_index].InUse := TRUE;
	            #sa_Parameter[#ti_index].RamOnly := FALSE;
	        END_REGION

	        REGION Step 34 - P560 Save [0..2]
	            #ti_index := #ti_index + 1;
	            #sa_Parameter[#ti_index].ParaNumber := 560;
	            #sa_Parameter[#ti_index].Index := 0;
	            #sa_Parameter[#ti_index].WriteValue := 1; // 1= save RAM & EERPOM
	            #sa_Parameter[#ti_index].WriteAccess := TRUE;
	            #sa_Parameter[#ti_index].ParaSet := 0;
	            #sa_Parameter[#ti_index].Format32 := FALSE;
	            #sa_Parameter[#ti_index].ActualValue := 0;
	            #sa_Parameter[#ti_index].InUse := TRUE;
	            #sa_Parameter[#ti_index].RamOnly := FALSE;
	        END_REGION

	        REGION Step 35 - P550 Copy internal EEPROM to external EEPROM [0..3]
	            #ti_index := #ti_index + 1;
	            #sa_Parameter[#ti_index].ParaNumber := 550;
	            #sa_Parameter[#ti_index].Index := 0;
	            #sa_Parameter[#ti_index].WriteValue := 2; // 2 = Copy internal to external EEPROM
	            #sa_Parameter[#ti_index].WriteAccess := FALSE;
	            #sa_Parameter[#ti_index].ParaSet := 0;
	            #sa_Parameter[#ti_index].Format32 := FALSE;
	            #sa_Parameter[#ti_index].ActualValue := 0;
	            #sa_Parameter[#ti_index].InUse := TRUE;
	            #sa_Parameter[#ti_index].RamOnly := FALSE;
	        END_REGION
	    END_IF;

	    (* IF #ix_VFDReadyToRun AND #sx_24VCommissioningDone THEN
	         REGION Step 39 - P220 Measurement [0..2]
	             #ti_index := 0;
	             #sa_Parameter[#ti_index].ParaNumber := 220;
	             #sa_Parameter[#ti_index].Index := 0;
	             #sa_Parameter[#ti_index].WriteValue := 2; // 2 =  Motor identification
	             #sa_Parameter[#ti_index].WriteAccess := TRUE;
	             #sa_Parameter[#ti_index].ParaSet := 1;
	             #sa_Parameter[#ti_index].Format32 := FALSE;
	             #sa_Parameter[#ti_index].ActualValue := 0;
	             #sa_Parameter[#ti_index].InUse := TRUE;
	             #sa_Parameter[#ti_index].RamOnly := FALSE;
	         END_REGION

	         REGION Step 40 - P220 Read if measurement started
	             #ti_index := #ti_index + 1;
	             #sa_Parameter[#ti_index].ParaNumber := 220;
	             #sa_Parameter[#ti_index].Index := 0;
	             #sa_Parameter[#ti_index].WriteValue := 0;
	             #sa_Parameter[#ti_index].WriteAccess := FALSE;
	             #sa_Parameter[#ti_index].ParaSet := 1;
	             #sa_Parameter[#ti_index].Format32 := FALSE;
	             #sa_Parameter[#ti_index].ActualValue := 0;
	             #sa_Parameter[#ti_index].InUse := TRUE;
	             #sa_Parameter[#ti_index].RamOnly := FALSE;
	         END_REGION

	         REGION Step 41 - P220 Read if measurement finished
	             #ti_index := #ti_index + 1;
	             #sa_Parameter[#ti_index].ParaNumber := 220;
	             #sa_Parameter[#ti_index].Index := 0;
	             #sa_Parameter[#ti_index].WriteValue := 0;
	             #sa_Parameter[#ti_index].WriteAccess := FALSE;
	             #sa_Parameter[#ti_index].ParaSet := 1;
	             #sa_Parameter[#ti_index].Format32 := FALSE;
	             #sa_Parameter[#ti_index].ActualValue := 0;
	             #sa_Parameter[#ti_index].InUse := TRUE;
	             #sa_Parameter[#ti_index].RamOnly := FALSE;
	         END_REGION


	         REGION Step 42 - P560 Save [0..2] (Step 39 - without motor identification)
	             #ti_index := #ti_index + 1;
	             #sa_Parameter[#ti_index].ParaNumber := 560;
	             #sa_Parameter[#ti_index].Index := 0;
	             #sa_Parameter[#ti_index].WriteValue := 1; // 1= save RAM & EERPOM
	             #sa_Parameter[#ti_index].WriteAccess := TRUE;
	             #sa_Parameter[#ti_index].ParaSet := 0;
	             #sa_Parameter[#ti_index].Format32 := FALSE;
	             #sa_Parameter[#ti_index].ActualValue := 0;
	             #sa_Parameter[#ti_index].InUse := TRUE;
	             #sa_Parameter[#ti_index].RamOnly := FALSE;
	         END_REGION

	         REGION Step 43 - P550 Copy internal EEPROM to external EEPROM [0..3] (Step 40 - without motor identification)
	             #ti_index := #ti_index + 1;
	             #sa_Parameter[#ti_index].ParaNumber := 550;
	             #sa_Parameter[#ti_index].Index := 0;
	             #sa_Parameter[#ti_index].WriteValue := 2; // 2 = Copy internal to external EEPROM
	             #sa_Parameter[#ti_index].WriteAccess := FALSE;
	             #sa_Parameter[#ti_index].ParaSet := 0;
	             #sa_Parameter[#ti_index].Format32 := FALSE;
	             #sa_Parameter[#ti_index].ActualValue := 0;
	             #sa_Parameter[#ti_index].InUse := TRUE;
	             #sa_Parameter[#ti_index].RamOnly := FALSE;
	         END_REGION
	         #sx_MotorMeasurement := TRUE;

	     END_IF; *)

	    // END_IF;

	END_REGION

	REGION 3 - Cancel job

	    // Monitor falling trigger if is input enable signal
	    #sF_TRIG_CancelJob(CLK := #iqx_Enable);

	    IF (#sF_TRIG_CancelJob.Q)
	    THEN
	        // IF parametrization is NOT done
	        IF (NOT #sx_Done)
	        THEN

	            #sx_Error := TRUE;
	            #sx_ReadOrder := FALSE;
	            #sx_WriteOrder := FALSE;
	            #sFB_ParaAcycWrite.qx_Done := FALSE;
	            #sx_Start := FALSE;
	            #sx_Busy := FALSE;

	        END_IF;

	    END_IF;

	END_REGION

	REGION 4 - Caclulaton used step in the sequence
	    // If maximum step is not calculated and input enable signal
	    IF (NOT #sx_MaxStepCalculation
	        AND #iqx_Enable)
	    THEN

	        // Create loop from maximum step number = 1 to 80
	        FOR #si_StepMax := 1 TO 80 DO

	            IF (NOT #sa_Parameter[#si_StepMax].InUse)   // If step commissioning is not used in sequence
	            THEN
	                #sx_MaxStepCalculation := TRUE;
	                EXIT;
	            END_IF;
	        END_FOR;
	    END_IF;
	END_REGION

	REGION 5 - Prepare data

	    IF (#sx_Start                                       // If occurs: signal to start of parametrization
	        AND NOT #sx_PreparedData                        // And step data is not prepared
	        AND NOT #sa_Status.StepDone                      // And parametrization is not done
	        AND #iqx_Enable)                                // And input enable signal
	    THEN

	        #sx_WriteOrder := #sa_Parameter[#sa_Status.StepNr].WriteAccess;
	        #sx_ReadOrder := NOT #sa_Parameter[#sa_Status.StepNr].WriteAccess;
	        #sx_PreparedData := TRUE;

	    END_IF;
	END_REGION

	REGION 6 - Call write parameter block

	    IF #sx_WriteOrder AND #sx_PreparedData THEN
	        #sFB_ParaAcycWrite(HW_Identifier := #ihw_HardwareID,
	                           idi_Value := #sa_Parameter[#sa_Status.StepNr].WriteValue,
	                           ii_ParameterNumber := #sa_Parameter[#sa_Status.StepNr].ParaNumber,
	                           ii_ParameterIndex := #sa_Parameter[#sa_Status.StepNr].Index,
	                           ii_ParameterSet := #sa_Parameter[#sa_Status.StepNr].ParaSet,
	                           ix_Parameter32Bit := #sa_Parameter[#sa_Status.StepNr].Format32,
	                           ix_RAM_Only := #sa_Parameter[#sa_Status.StepNr].RamOnly,
	                           ix_Execute := NOT #sFB_ParaAcycWrite.qx_Done,
	                           qx_Done => #sFB_ParaAcycWrite.qx_Done,
	                           qx_Busy => #sFB_ParaAcycWrite.qx_Busy,
	                           qx_Error => #sFB_ParaAcycWrite.qx_Error,
	                           qdi_ValueRead => #sa_Parameter[#sa_Status.StepNr].ActualValue,
	                           qw_ErrorID => #sFB_ParaAcycWrite.qw_ErrorID);

	        #sR_TRIG_Done(CLK := #sFB_ParaAcycWrite.qx_Done);
	    END_IF;
	END_REGION

	REGION 7 - Call read parameter block

	    IF #sx_ReadOrder AND #sx_PreparedData THEN
	        #sFB_ParaAcycRead(iHW_Identifier := #ihw_HardwareID,
	                          ix_Enable := TRUE,
	                          ii_Parameter_Number := #sa_Parameter[#sa_Status.StepNr].ParaNumber,
	                          ii_Parameter_Index := #sa_Parameter[#sa_Status.StepNr].Index,
	                          ii_Parameter_Set := #sa_Parameter[#sa_Status.StepNr].ParaSet,
	                          qx_Valid => #sFB_ParaAcycRead.qx_Valid,
	                          qx_Busy => #sFB_ParaAcycRead.qx_Busy,
	                          qx_Error => #sFB_ParaAcycRead.qx_Error,
	                          qw_Error_ID => #sFB_ParaAcycRead.qw_Error_ID,
	                          qdi_Value => #sFB_ParaAcycRead.qdi_Value);
	    END_IF;
	END_REGION

	REGION 8 - Status commissioning

	    REGION 8.1 Step number error

	        IF (#sx_WriteOrder AND #sFB_ParaAcycWrite.qx_Error)
	            OR
	            (#sx_ReadOrder AND #sFB_ParaAcycRead.qx_Error)
	            OR #sa_Status.TimeExceeded
	        THEN
	            #sx_Start := FALSE;
	            #sx_Error := TRUE;
	            #sx_Done := FALSE;

	            #sx_WriteOrder := FALSE;
	            #sx_ReadOrder := False;
	            #sa_Status.StepNrError := #sa_Status.StepNr;
	        END_IF;
	    END_REGION


	    REGION 8.2 - Read done

	        IF #sx_ReadOrder
	            AND NOT #sFB_ParaAcycRead.qx_Busy
	            AND NOT #sFB_ParaAcycRead.qx_Error
	            AND #sFB_ParaAcycRead.qx_Valid

	        THEN

	            #sa_Status.StepDone := TRUE;
	            #sx_ReadOrder := FALSE;
	            #sa_Parameter[#sa_Status.StepNr].ActualValue := DINT_TO_INT(#sFB_ParaAcycRead.qdi_Value);

	            IF #sa_Parameter[#sa_Status.StepNr].ParaNumber = 846
	            THEN
	                #qi_HWAdress := DINT_TO_INT(#sFB_ParaAcycRead.qdi_Value);
	            END_IF;

	        END_IF;
	    END_REGION


	    REGION 8.3 - Write done

	        IF #sx_WriteOrder
	            AND NOT #sFB_ParaAcycWrite.qx_Error
	            AND #sR_TRIG_Done.Q
	        THEN
	            #sa_Status.StepDone := TRUE;
	            #sx_WriteOrder := FALSE;
	            #sFB_ParaAcycWrite.qx_Done := FALSE;
	        END_IF;
	    END_REGION

	    REGION 8.4 - Step time watchdog
	        // the function is too long active
	        IF #iqx_Enable AND "DB_Memory"."OS_0.1sec"
	        THEN
	            #si_StepTime += 1;
	        END_IF;
	        IF (#si_StepTime > #ci_MaxStepTime)
	        THEN
	            #sa_Status.TimeExceeded := TRUE;
	        ELSE
	            #sa_Status.TimeExceeded := FALSE;
	        END_IF;
	    END_REGION
	END_REGION

	REGION 9 - Go to next step

	    IF #iqx_Enable
	        AND #sa_Status.StepDone
	        AND "DB_Memory".OS_2sec
	    THEN
	        #sx_PreparedData := FALSE;
	        #sa_Status.StepDone := FALSE;
	        #sa_Status.StepNr += 1;
	        #si_StepTime := 0;
	    END_IF;
	END_REGION

	REGION 10 - Commissioning done

	    IF (#si_StepMax <= #sa_Status.StepNr
	        AND #iqx_Enable)
	    THEN
	        #iqx_Enable := FALSE;
	        #sx_Done := TRUE;
	        #sx_Start := FALSE;
	        #sx_Busy := FALSE;
	        #sx_24VCommissioningDone := TRUE;

	    END_IF;
	END_REGION

	REGION 11 - Write output

	    #qx_Busy := #sx_Busy;
	    #qx_Done := #sx_Done;
	    #qx_Error := #sx_Error;
	    #qx_24VCommissioningDone := #sx_24VCommissioningDone;

	END_REGION


END_FUNCTION_BLOCK

TYPE "UDT_CognexDM260_IN"
VERSION : 0.1
   STRUCT
      TriggerReady : Bool;   // Indicates when the device is ready to accept a new trigger. Bit is True when “Trigger Enable”is set and the device is ready to accept a new trigger.
      TriggerAck : Bool;   // Indicates that the DataMan has received a new Trigger. This bit remains True as long as the“Trigger” bit remains True (that is, it is interlocked with the Trigger bit).
      "Acquiring/Reserved??" : Bool;   // Reserved for future use.
      MissedAcq : Bool;   // Indicates that the DataMan was unable to successfully trigger an acquisition. Bit is cleared
      "Not used" : Bool;   // Reserved for future use.8-23
      "Not used_1" : Bool;   // Reserved for future use.8-23
      "Not used_2" : Bool;   // Reserved for future use.8-23
      "Not used_3" : Bool;   // Reserved for future use.8-23
      TriggerID : Byte;   // HIGHER BYTE ID value of the next trigger to be issued (16-bit integer). Used to match issued triggers withcorresponding result data received later. This same value is returned in ResultID of theresult data.
      "TriggerID 1" : Byte;   // LOWER BYTE ID value of the next trigger to be issued (16-bit integer). Used to match issued triggers withcorresponding result data received later. This same value is returned in ResultID of theresult data.
      BYTE_Decoding : Byte;   // Bit:0-Decode Complete, 1-Decode Complete, 2- Results Buffer Overrun, 3- Results Available, 4-6 Unused, 7 - General Fault
      "Train Code Ack" : Bool;   // Indicates that the “Train Code” operation is complete
      "Train Match String Ack" : Bool;   // Indicates that the “Train Match String” operation is complete
      "Train Focus Ack" : Bool;   // Indicates that the “Train Focus” operation is complete
      "Train Brightness Ack" : Bool;   // Indicates that the “Train Brightness” operation is complete
      "Untrain Ack" : Bool;   // Indicates that the “Untrain” operation is complete
      Reserved : Bool;   // Reserved for future use
      "Execute DMCC Ack" : Bool;   // Indicates that the “Execute DMCC” operation is complete
      "Set Match String Ack" : Bool;   // Indicates that the “Set Match String” operation is complete - User Data Option - Currently only used by “Set Match String” soft event.
      ResultID : Byte;   // HIGHER BYTE The value of the “Trigger ID” when the trigger that generated these results was issued. Used to match up triggers with corresponding result data (16-bit Integer).
      "ResultID 1" : Byte;   // LOWER BYTE The value of the “Trigger ID” when the trigger that generated these results was issued. Used to match up triggers with corresponding result data (16-bit Integer).
      "Result Code" : Byte;   // HIGHER BYTE not used
      "Result Code_1" : Byte;   // Indicates the success or failure of the read that produced these results (16-bit Integer).Bit 0,1=read, 0=no read, Bit 1,1=validated, 0=not validated (or validation not in use),  Bit 2,1=verified, 0=not verified (or verification not in use)  Bit 3,1=acquisition trigger overrun  Bit 4,1=acquisition buffer overflow
      "Result Extended" : Byte;   // Currently unused (16-bit Integer).
      "Result Extended_1" : Byte;   // Currently unused (16-bit Integer).
      "Result Length" : Byte;   // HIGHER BYTE Actual number of bytes of read data contained in the “Result Data” field (16-bitInteger).
      "Result Length_1" : Byte;   // LOWER BYE Actual number of bytes of read data contained in the “Result Data” field (16-bitInteger).
      "BarCodeValue[0]-NO_READ_sign" : Char;   // First barecode char
      BarCodeValue : Array[1..63] of Char;   // Remaining characters of the barcode, after the barcode remaining chars are  '$00' = BYTE#16#00
   END_STRUCT;

END_TYPE

FUNCTION_BLOCK "FB_ParcelLength"
{ S7_Optimized_Access := 'TRUE' }
VERSION : 0.1
// ATTRIBUTES
// AUTO_NUMBER = True
// BLOCK_NUMBER = 20
// END_ATTRIBUTES
   VAR_INPUT
      ii_PECPosition { ExternalAccessible := 'False'; ExternalVisible := 'False'; ExternalWritable := 'False'} : Int;   //    Photoeye position [cm]
      ii_Displacement { ExternalAccessible := 'False'; ExternalVisible := 'False'; ExternalWritable := 'False'} : Int;   //    Displacement [cm]
      ix_LengthMeasurementEnable { ExternalAccessible := 'False'; ExternalVisible := 'False'; ExternalWritable := 'False'} : Bool;   //    Length measurement enable
      ix_GapMeasurementEnable { ExternalAccessible := 'False'; ExternalVisible := 'False'; ExternalWritable := 'False'} : Bool;   //    Gap measurement enable
   END_VAR

   VAR_IN_OUT
      iqa_TrackingData : Array[*] of Int;   //    Tracking data
   END_VAR

   VAR
      sR_TRIG_Data {InstructionName := 'R_TRIG'; LibVersion := '1.0'; ExternalAccessible := 'False'; ExternalVisible := 'False'; ExternalWritable := 'False'; S7_SetPoint := 'False'} : R_TRIG;   //    Data rising edge for length and gap measurements
      sF_TRIG_Data {InstructionName := 'F_TRIG'; LibVersion := '1.0'; ExternalAccessible := 'False'; ExternalVisible := 'False'; ExternalWritable := 'False'; S7_SetPoint := 'False'} : F_TRIG;   //    Data falling edge for length and gap measurements
      si_Length { ExternalAccessible := 'False'; ExternalVisible := 'False'; ExternalWritable := 'False'} : Int;   //    Parcel length
      si_Gap { ExternalAccessible := 'False'; ExternalVisible := 'False'; ExternalWritable := 'False'} : Int;   //    Gap distance
      si_GIN { ExternalAccessible := 'False'; ExternalVisible := 'False'; ExternalWritable := 'False'} : Int;   //    GIN number of current measured parcel
      si_OldGIN { ExternalAccessible := 'False'; ExternalVisible := 'False'; ExternalWritable := 'False'} : Int;   //    GIN number of previous mesured parcel
   END_VAR

   VAR CONSTANT
      ci_Overflow : Int := 32767;   //    Integer overflow value
   END_VAR


BEGIN
	(*
	----------------------------------------------------------------------------------------

	Version history:
	Date        | Version   | Author        | Remark
	----------------------------------------------------------------------------------------
	21/02/2020  | 3.1       | L.Klar        | first release MHSE TIA 15.1
	21/02/2023  | 4.0       | F.Baten       | 4.0 Release TIA 17.5
	*)

	REGION 1 – Data triggers

	    // Triggers to detect front and end of data

	    #sR_TRIG_Data(CLK := #iqa_TrackingData[#ii_PECPosition] > 0);
	    #sF_TRIG_Data(CLK := #iqa_TrackingData[#ii_PECPosition] > 0);

	END_REGION

	REGION 2 – Length counter

	    //  Length is counted from a displacement, when data is available
	    //
	    IF (#iqa_TrackingData[#ii_PECPosition] > 0
	        AND #ix_LengthMeasurementEnable
	        AND #si_Length < #ci_Overflow)

	    THEN
	        #si_Length += #ii_Displacement;
	    END_IF;

	END_REGION

	REGION 3 – Gap counter

	    //  Gap is counted from a displacement, when data isn't available
	    IF (#iqa_TrackingData[#ii_PECPosition] = 0
	        AND #ix_GapMeasurementEnable
	        AND #si_Gap < #ci_Overflow)
	    THEN
	        #si_Gap += #ii_Displacement;
	    END_IF;

	END_REGION

	REGION 4 – Parcel GIN

	    IF (#sR_TRIG_Data.Q AND
	        (#ix_LengthMeasurementEnable OR #ix_GapMeasurementEnable))
	    THEN
	        #si_GIN := #iqa_TrackingData[#ii_PECPosition];
	    END_IF;

	END_REGION

	REGION 5 – Write length into a GIN record

	    IF (#sF_TRIG_Data.Q)
	    THEN

	        IF #ix_LengthMeasurementEnable OR #ix_GapMeasurementEnable THEN
	            #si_OldGIN := #si_GIN;
	        END_IF;

	        IF (#si_GIN > 0
	            AND ABS(#si_Length) > 0
	            AND #ix_LengthMeasurementEnable)
	        THEN
	            "DB_GIN".GIN[#si_GIN].General.Length := ABS(#si_Length) - 1;
	            #si_Length := 0;
	        ELSE
	            #si_Length := 0;
	        END_IF;
	    END_IF;

	END_REGION

	REGION 6 – Write GIN into a GIN record

	    IF (#sR_TRIG_Data.Q)
	    THEN
	        IF (#si_OldGIN > 0
	            AND #si_GIN > 0
	            AND #si_Gap <> 0
	            AND #si_OldGIN <> #si_GIN
	            AND #ix_GapMeasurementEnable)
	        THEN
	            IF (#ii_Displacement > 0)
	            THEN
	                "DB_GIN".GIN[#si_GIN].General.LeadingGap := ABS(#si_Gap) - 1;
	                "DB_GIN".GIN[#si_OldGIN].General.TrailingGap := "DB_GIN".GIN[#si_GIN].General.LeadingGap;
	                #si_Gap := 0;
	            ELSIF (#ii_Displacement < 0)
	            THEN
	                "DB_GIN".GIN[#si_OldGIN].General.LeadingGap := ABS(#si_Gap - 1);
	                "DB_GIN".GIN[#si_GIN].General.TrailingGap := "DB_GIN".GIN[#si_OldGIN].General.LeadingGap;
	                #si_Gap := 0;
	            END_IF;
	        ELSE
	            #si_Gap := 0;
	        END_IF;
	    END_IF;

	END_REGION
END_FUNCTION_BLOCK

TYPE "UDT_DataLogicBlade_IN_SN"
VERSION : 0.1
   STRUCT
      Data : Array[0..15] of Byte;
   END_STRUCT;

END_TYPE

TYPE "UDT_CommisioningNord"
VERSION : 0.1
   STRUCT
      HWAdress : Int;   // Actual dipswitch adress of the VFD
      i_ParCRC : Word;   // VFD generated CRC
      CommissionError { ExternalAccessible := 'False'; ExternalVisible := 'False'; ExternalWritable := 'False'} : Bool;   // Commissioning error active
   END_STRUCT;

END_TYPE

TYPE "UDT_StatusTC36"
VERSION : 0.1
//One direction, motor, controler, EOS
   STRUCT
      RightAngledTransfer : "UDT_RATStatus";   // Right angled transfer status
      MCO_M01 : "UDT_AixControllerStatus";   // MCO Status
   END_STRUCT;

END_TYPE

TYPE "UDT_CognexDM260_OUT"
VERSION : 0.1
   STRUCT
      TriggerEnable : Bool;   // Setting this bit enables triggering via PROFINET. Clearing this bit disables triggering.
      Trigger : Bool;   // Setting this bit triggers an acquisition when the following conditions are met:l Trigger Enable is set.l No acquisition is currently in progress.l The device is ready to trigger.
      Reserved_0 : Bool;   // Reserved for future use
      Reserved_1 : Bool;   // Reserved for future use
      Reserved_2 : Bool;   // Reserved for future use
      Reserved_3 : Bool;   // Reserved for future use
      Reserved_4 : Bool;   // Reserved for future use
      Reserved_5 : Bool;   // Reserved for future use
      BufferResultsEnable : Bool;   // Enables queuing of “Result Data”. If enabled, the current result data will remain until acknowledged (even if new results arrive). New results are queued. The reader can buffer up to 50 and the base station can buffer up to 500 sets of read results.
      ResultsAck : Bool;   // Bit is used to acknowledge that the PLC has successfully read the latest result data. When set True the “Result Available” bit will be cleared. If result buffering is enabled, the next set of result data will be pulled from the queue and “Result Available” will again be set True.
      Reserved : Bool;   // Reserved for future use.
      Reserved_1_1 : Bool;   // Reserved for future use.
      Reserved_2_1 : Bool;   // Reserved for future use.
      Reserved_3_1 : Bool;   // Reserved for future use.
      Reserved_4_1 : Bool;   // Reserved for future use.
      Reserved_5_1 : Bool;   // Reserved for future use.
      "Train Code" : Bool;   // Bit transition from 0 -> 1 causes the train code operation to be invoked.
      "Train Match String" : Bool;   // Bit transition from 0 -> 1 causes the train match string operation to be invoked.
      "Train Focus" : Bool;   // Bit transition from 0 -> 1 causes the train focus operation to be invoked.
      "Train Brightness" : Bool;   // Bit transition from 0 -> 1 causes the train brightness operation to be invoked
      Untrain : Bool;   // Bit transition from 0 -> 1 causes the untrain operation to be invoked.
      Reserved_6 : Bool;   // Reserved for future use
      "Execute DMCC" : Bool;   // Bit transition from 0 -> 1 causes the DMCC operation to be invoked. Note that a valid DMCC command string must first be placed in “User Data” before invoking this event.
      "Set Match String" : Bool;   // Bit transition from 0 -> 1 causes the set match string operation to be invoked. Note that match string data must first be placed in “User Data” before invoking this event.
      "UserData Option" : Int;   // Specifies which code target to assign the string (16-bit Integer). 1, assign string to 2D codes, 2, assign string to QR codes
      "UserData Length" : Int;   // Number of bytes of valid data actually contained in the “User Data” field (16-bit
      "UserData[0]" : Byte;   // Data sent from the PLC to the DataMan to support acquisition, decoding, andother special operations (array of bytes). User Data Option - Currently only used by “Set Match String” soft event.
      "UserData[1]" : Byte;
      "UserData[2]" : Byte;
      "UserData[3]" : Byte;
      "UserData[4]" : Byte;
      "UserData[5]" : Byte;
      "UserData[6]" : Byte;
      "UserData[7]" : Byte;
      "UserData[8]" : Byte;
      "UserData[9]" : Byte;
      "UserData[10]" : Byte;
      "UserData[11]" : Byte;
      "UserData[12]" : Byte;
      "UserData[13]" : Byte;
      "UserData[14]" : Byte;
      "UserData[15]" : Byte;
      "UserData[16]" : Byte;
      "UserData[17]" : Byte;
      "UserData[18]" : Byte;
      "UserData[19]" : Byte;
      "UserData[20]" : Byte;
      "UserData[21]" : Byte;
      "UserData[22]" : Byte;
      "UserData[23]" : Byte;
      "UserData[24]" : Byte;
      "UserData[25]" : Byte;
      "UserData[26]" : Byte;
      "UserData[27]" : Byte;
      "UserData[28]" : Byte;
      "UserData[29]" : Byte;
      "UserData[30]" : Byte;
      "UserData[31]" : Byte;
      "UserData[32]" : Byte;
      "UserData[33]" : Byte;
      "UserData[34]" : Byte;
      "UserData[35]" : Byte;
      "UserData[36]" : Byte;
      "UserData[37]" : Byte;
      "UserData[38]" : Byte;
      "UserData[39]" : Byte;
      "UserData[40]" : Byte;
      "UserData[41]" : Byte;
      "UserData[42]" : Byte;
      "UserData[43]" : Byte;
      "UserData[44]" : Byte;
      "UserData[45]" : Byte;
      "UserData[46]" : Byte;
      "UserData[47]" : Byte;
      "UserData[48]" : Byte;
      "UserData[49]" : Byte;
      "UserData[50]" : Byte;
      "UserData[51]" : Byte;
      "UserData[52]" : Byte;
      "UserData[53]" : Byte;
      "UserData[54]" : Byte;
      "UserData[55]" : Byte;
      "UserData[56]" : Byte;
      "UserData[57]" : Byte;
      "UserData[58]" : Byte;
      "UserData[59]" : Byte;
      "UserData[60]" : Byte;
      "UserData[61]" : Byte;
      "UserData[62]" : Byte;
      "UserData[63]" : Byte;
   END_STRUCT;

END_TYPE

TYPE "UDT_StatusTC13"
VERSION : 0.1
//One direction, motor, controler, EOS, Tracking
//
   STRUCT
      Conveyor : "UDT_ConveyorStatus";   // Conveyor Status
      PEC_EoS : "UDT_PECUpdateStatus";   // PEC EoS Status
      MCO_M01 : "UDT_AixControllerStatus";   // MCO Status
   END_STRUCT;

END_TYPE

TYPE "UDT_VfdSEWPositioningPO"
TITLE = UDT_VFD_SEW_PO
VERSION : 0.1
//User-defined structure of VFD SEW output telegram.
   STRUCT
      Control_Word_1 : Struct   // Control Word 1
         ResetError { ExternalAccessible := 'False'; ExternalVisible := 'False'; ExternalWritable := 'False'} : Bool;   // Reset error "1"
         BIT_09_Reserved { ExternalAccessible := 'False'; ExternalVisible := 'False'; ExternalWritable := 'False'} : Bool;   // Reserved
         ActivateDriveTrain2 { ExternalAccessible := 'False'; ExternalVisible := 'False'; ExternalWritable := 'False'} : Bool;   // Activate drive train 2 "1"
         BIT_11_Reserved { ExternalAccessible := 'False'; ExternalVisible := 'False'; ExternalWritable := 'False'} : Bool;   // Reserved
         DeactivateSW_LimitSwitch { ExternalAccessible := 'False'; ExternalVisible := 'False'; ExternalWritable := 'False'} : Bool;   // Deactivate software limit switch "1"
         ActivateInhibit { ExternalAccessible := 'False'; ExternalVisible := 'False'; ExternalWritable := 'False'} : Bool;   // Activate inhibit "1"
         ActivateStandby { ExternalAccessible := 'False'; ExternalVisible := 'False'; ExternalWritable := 'False'} : Bool;   // Activate standby "1"
         MovikitHandshakeIn { ExternalAccessible := 'False'; ExternalVisible := 'False'; ExternalWritable := 'False'} : Bool;   // If the MOVIKIT works the value will be copied into "MovikitHandshakeOut"
         EnableRapidStop { ExternalAccessible := 'False'; ExternalVisible := 'False'; ExternalWritable := 'False'} : Bool;   // Enable “1” / Rapid stop “0”
         EnableApplicationStop { ExternalAccessible := 'False'; ExternalVisible := 'False'; ExternalWritable := 'False'} : Bool;   // Enable “1” / Application stop “0”
         BIT_02_Reserved { ExternalAccessible := 'False'; ExternalVisible := 'False'; ExternalWritable := 'False'} : Bool;   // Reserved
         ReleaseBrake { ExternalAccessible := 'False'; ExternalVisible := 'False'; ExternalWritable := 'False'} : Bool;   // Release brake "1"
         JogPos { ExternalAccessible := 'False'; ExternalVisible := 'False'; ExternalWritable := 'False'} : Bool;   // Jog in positive direction "1"
         JogNeg { ExternalAccessible := 'False'; ExternalVisible := 'False'; ExternalWritable := 'False'} : Bool;   // Jog in negative direction "1"
         ApplyRelativePositioning { ExternalAccessible := 'False'; ExternalVisible := 'False'; ExternalWritable := 'False'} : Bool;   // Take the relative position from the FCB09 "1"
         StartStop { ExternalAccessible := 'False'; ExternalVisible := 'False'; ExternalWritable := 'False'} : Bool;   // Start "1" / Stop "0"
      END_STRUCT;
      SetpointSpeed : Int;   // Speed (Int) [mm/s]
      SetpointAcceleration : Int;   // Acceleration (Int) [mm/s²]
      SetpointDeceleration : Int;   // Decceleration (Int) [mm/s²]
      DigitalOutputs : Word;   // Digital Outputs
      SetpointMode : Int;   // Set the application mode (Int)
      SetpointPosition_hW : Word;   // Setpoint Position - High Word
      SetpointPosition_lW : Word;   // Setpoint Position - Low Word
   END_STRUCT;

END_TYPE

TYPE "UDT_RIOVSUStatistics"
TITLE = UDT_RIOStatistics
VERSION : 0.1
//User-defined structure of FB_RIO function block statistics.
   STRUCT
      Int400VCBError : "UDT_EventStatistic";   // Statistics of internal 400V circuit breaker not OK
      Ext400VError : "UDT_EventStatistic";   // Statistics of external 400V not OK
      "24VError" : "UDT_EventStatistic";   // Statistics of external 24V not OK
      BrakeCBerror : "UDT_EventStatistic";   // Statistics of brake circuit breaker not OK
      BrakeThermError : "UDT_EventStatistic";   // Statistics of brake thermal error
      PNSlaveNotOnline : "UDT_EventStatistic";   // Statistics of Profinet slave not online
      PNSlaveError : "UDT_EventStatistic";   // Statistics of a Profinet slave error
   END_STRUCT;

END_TYPE

TYPE "UDT_VfdStatus"
TITLE = UDT_VfdStatus
VERSION : 0.1
//User-defined structure of VFD status.
   STRUCT
      ErrorCode : Int;   // Error code
      SubErrorCode : Int;   // Sub error code
      PNSlaveNotonline : Bool := FALSE;   // Profinet slave is not on line
      PNSlaveError : Bool := FALSE;   // Profinet slave has an error
      InternalError : Bool := FALSE;   // A VFD internal error is active, see error code
      InternalWarning : Bool := FALSE;   // A VFD internal warning is active, see error code
      CommunicationErrorMovikit : Bool := FALSE;   // Communication error with MoviKit
      VFDRunningFeedbackError : Bool := FALSE;   // Motor is not running
      PNSlaveWarning { ExternalAccessible := 'False'; ExternalVisible := 'False'; ExternalWritable := 'False'} : Bool;   // Profinet slave has a warning
   END_STRUCT;

END_TYPE

TYPE "UDT_VSULiftStatus"
TITLE = UDT_VSUStatus
VERSION : 0.1
//User-defined structure of FB_VerticalSwitch function block status.
   STRUCT
      Status { ExternalWritable := 'False'} : Int;   // Status number
      Specific { ExternalWritable := 'False'} : Struct   // Equipment specific warnings and errors
         ReferencedErr { ExternalWritable := 'False'} : Bool;   // VFD is not referenced
         ExitGapErr { ExternalWritable := 'False'} : Bool;   // Exit gap check was activated when moving
         EntryGapErr { ExternalWritable := 'False'} : Bool;   // Entrance gap check was activated when moving
         BeltTear1Err { ExternalWritable := 'False'} : Bool;   // Belt tear detected - Sensor 1
         BeltTear2Err { ExternalWritable := 'False'} : Bool;   // Belt tear detected - Sensor 2
         MaintSupport1Err { ExternalWritable := 'False'} : Bool;   // Maintenace support 1 extracted in automatic mode
         MaintSupport2Err { ExternalWritable := 'False'} : Bool;   // Maintenace support 2 extracted in automatic mode
         UpperPositionErr { ExternalWritable := 'False'} : Bool;   // Upper position overrun
         LowerPositionErr { ExternalWritable := 'False'} : Bool;   // Lower position overrun
         DirectionErr { ExternalWritable := 'False'} : Bool;   // Item in the wrong position
         KeyswitchWrn { ExternalWritable := 'False'} : Bool;   // Keyswitch is in '0' position
         SafetyDoorDownErr { ExternalWritable := 'False'} : Bool;   // Safety door down diagnostic fault
         SafetyDoorUpErr { ExternalWritable := 'False'} : Bool;   // Safety door up diagnostic fault
         LiftKeySwitchStop { ExternalWritable := 'False'} : Bool;   // Lift key switch turned to Stop
         MaintenanceSwitchUp { ExternalWritable := 'False'} : Bool;
      END_STRUCT;
   END_STRUCT;

END_TYPE

TYPE "UDT_StatisticsTC11"
VERSION : 0.1
//One direction, motor
   STRUCT
      Conveyor : "UDT_ConveyorStatistics";   // Conveyor Statistics
      MCO_M01 : "UDT_VfdStatistics";   // MCO Statistics
   END_STRUCT;

END_TYPE

FUNCTION "FC_GetPNPortStatus" : Void
{ S7_Optimized_Access := 'TRUE' }
VERSION : 0.1
// ATTRIBUTES
// AUTO_NUMBER = True
// BLOCK_NUMBER = 20
// END_ATTRIBUTES
   VAR_INPUT
      ii_NumberOfPorts : Int;   //  Number of ports in device
      iUDT_DevicePNInfo : "UDT_PNDevice";   //  PN device info structure
   END_VAR

   VAR_OUTPUT
      qa_PortFault : Array[1..8] of Bool;   //  When TRUE then specific port has a fault
   END_VAR

   VAR_TEMP
      tp_GetDiagInfo {InstructionName := 'DIS'; LibVersion := '1.0'} : DIS;   //  Diagnostic structure
      tp_DeviceGeoAddr {InstructionName := 'GEOADDR'; LibVersion := '1.0'} : GEOADDR;   //  Device pointer structre
      ta_PortFault : Array[1..8] of Bool;   //  When TRUE then port has a fault
      ti_Geo2LogStatus : Int;   //  GEO2LOG status code
      ti_GetDiagStatus : Int;   //  Get_Diag status code
      ti_Log2GeoStatus : Int;   //  LOG2GEO status code
      ti_Loopcounter : Int;   //  Loop counter
      tui_cnt : UInt;   //  Not used
      tdi_PortLaddr : HW_ANY;   //  HW identifier
      ti_PortFault : Bool;   //  At least one port is faulty
      tx_ConfigurationError : Bool;   //  Configuration error occurred
   END_VAR

   VAR CONSTANT
      ci_Area : UInt := 1;   //     Area ID of IO Profinet devices
      ci_HWTYPE : UInt := 5;
      ci_PortSlot : UInt := 0;
      ci_PortSubslot : Word := 16#8000;
   END_VAR


BEGIN
	(*
	----------------------------------------------------------------------------------------

	Version history:
	Date        | Version   | Author        | Remark
	----------------------------------------------------------------------------------------
	03/11/2020  | 3.0       | K.Pokorski    | first release MHS TIA 15.1
	17/12/2020  | 3.1       | K.Pokorski    | Run operation only during error
	21/02/2023  | 4.0       | F.Baten       | 4.0 Release TIA 17.5
	*)

	REGION 1 - Check configuration

	    #tx_ConfigurationError := #ii_NumberOfPorts < 1
	    OR #ii_NumberOfPorts > 8
	    OR NOT #iUDT_DevicePNInfo.PNDeviceFound;

	END_REGION

	REGION 2 - Read profinet network number

	    // Using LOG2GEO profinet network address is read
	    #ti_Log2GeoStatus := LOG2GEO(LADDR := "DB_ProfinetDiagnostic".ProfinetNetworks[#iUDT_DevicePNInfo.PNNetworknumber].DeviceStatus[#iUDT_DevicePNInfo.PNDeviceNumber].DeviceState.HW_ID,
	                                 GEOADDR := #tp_DeviceGeoAddr);

	END_REGION

	REGION 3 - Preparation the device pointer

	    // HWTYPE = 5 - Submodule
	    #tp_DeviceGeoAddr.HWTYPE := #ci_HWTYPE;
	    // AREA = 1 - PROFINET IO
	    #tp_DeviceGeoAddr.AREA := #ci_Area;
	    // SLOT = 0 - Ports are on slot 0
	    #tp_DeviceGeoAddr.SLOT := #ci_PortSlot;
	    // STATION - Profinet number
	    #tp_DeviceGeoAddr.STATION := "DB_ProfinetDiagnostic".ProfinetNetworks[#iUDT_DevicePNInfo.PNNetworknumber].DeviceStatus[#iUDT_DevicePNInfo.PNDeviceNumber].DeviceState.ProfinetNumber;

	END_REGION

	REGION 4 - Checking the port status
	    // If device report error and is available on the PN network
	    IF "DB_ProfinetDiagnostic".ProfinetNetworks[#iUDT_DevicePNInfo.PNNetworknumber].DeviceStatus[#iUDT_DevicePNInfo.PNDeviceNumber].DeviceState.Error
	        AND "DB_ProfinetDiagnostic".ProfinetNetworks[#iUDT_DevicePNInfo.PNNetworknumber].DeviceStatus[#iUDT_DevicePNInfo.PNDeviceNumber].DeviceState.Exist
	        AND NOT #tx_ConfigurationError
	    THEN

	        // Loop through all profinet ports
	        FOR #ti_Loopcounter := 1 TO #ii_NumberOfPorts DO
	            // Reset auxiliary port fault bit
	            #ta_PortFault[#ti_Loopcounter] := FALSE;
	            // SUBSLOT = 16#8000 plus port number (TIA structure to refer to port)
	            #tp_DeviceGeoAddr.SUBSLOT := INT_TO_UINT(WORD_TO_INT(#ci_PortSubslot) + (#ti_Loopcounter));
	            // Using GEO2LOG port address is read
	            #ti_Geo2LogStatus := GEO2LOG(GEOADDR := #tp_DeviceGeoAddr, LADDR => #tdi_PortLaddr);
	            // Using GET_DIAG port status is read
	            #ti_GetDiagStatus := GET_DIAG(MODE := 1, LADDR := #tdi_PortLaddr, CNT_DIAG => #tui_cnt, DIAG := #tp_GetDiagInfo);

	            // Set port fault if all operations do not report any error and port is faulty
	            IF #ti_GetDiagStatus = 0
	                AND #ti_Geo2LogStatus = 0
	                AND #ti_Log2GeoStatus = 0
	                AND #tp_GetDiagInfo.OwnState = 4
	            THEN
	                #ta_PortFault[#ti_Loopcounter] := TRUE;
	            END_IF;
	        END_FOR;
	        // Reset module status if error occurred
	    ELSIF #tx_ConfigurationError
	    THEN
	        FOR #ti_Loopcounter := 1 TO 8 DO
	            #ta_PortFault[#ti_Loopcounter] := FALSE;
	        END_FOR;
	    END_IF;

	END_REGION

	REGION 5 - Write output

	    #qa_PortFault := #ta_PortFault;

	END_REGION


END_FUNCTION

FUNCTION "FC_GetDevicePN" : Void
TITLE = FC_GetDevicePN
{ S7_Optimized_Access := 'TRUE' }
AUTHOR : MHSE
VERSION : 3.0
// ATTRIBUTES
// AUTO_NUMBER = True
// BLOCK_NUMBER = 18
// END_ATTRIBUTES
   VAR_INPUT
      is_PNDeviceName : String;   // Name of the device
      ix_SimulationModeActive : Bool;   // True = Simulation mode active
   END_VAR

   VAR_IN_OUT
      iqUDT_PND : "UDT_PNDevice";   // Device found in Profinet structure
   END_VAR

   VAR_TEMP
      ti_NrOfConfiguredPNNetworks : Int;   // Number of networks configured in project
      ti_NrOfDevices : Int;   // Nr of devices is networks
      ti_LcPNNetworkNumber : Int;   // Loop counter to find PN network number
      ti_LcPNDeviceNumber : Int;   // Loop counter to find PN device number
   END_VAR


BEGIN
	(*
	----------------------------------------------------------------------------------------

	Version history:
	Date        | Version   | Author        | Remark
	----------------------------------------------------------------------------------------
	16/09/2019  | 2.3       | F.Baten       | Cut out of 'FB_RIO'
	29/09/2019  | 2.4       | K.Pokorski    | Network seach started from 1 instead 0
	30/09/2019  | 2.5       | K.Pokorski    | Chagne prefixes of temporary varaibles from 'si' to 'ti'
	12/11/2019  | 3.0       | P.Majka       | 3.0 MHS library release TIA 15.1
	21/02/2023  | 4.0       | F.Baten       | 4.0 Release TIA 17.5
	*)

	REGION 1 - Get Device Profinet number
	    // if simulation is disabled
	    IF NOT #ix_SimulationModeActive
	    THEN
	        // And the profinet device is not found yet
	        IF (#is_PNDeviceName <> "DB_ProfinetDiagnostic".ProfinetNetworks[#iqUDT_PND.PNNetworknumber].DeviceStatus[#iqUDT_PND.PNDeviceNumber].DeviceState.PNDeviceName)
	            OR #iqUDT_PND.PNDeviceFound = FALSE
	        THEN
	            #iqUDT_PND.PNDeviceFound := FALSE;

	            // check how many profinet networks are configured
	            #ti_NrOfConfiguredPNNetworks := "FC_GetNrOfArrayEl"("DB_ProfinetDiagnostic".ProfinetNetworks);

	            FOR #ti_LcPNNetworkNumber := 1 TO (#ti_NrOfConfiguredPNNetworks) DO

	                #iqUDT_PND.PNNetworknumber := #ti_LcPNNetworkNumber;

	                // and check how many devices are configured per network
	                #ti_NrOfDevices := "FC_GetNrOfArrayEl"("DB_ProfinetDiagnostic".ProfinetNetworks[#iqUDT_PND.PNNetworknumber].DeviceStatus);

	                // check for each of the devices in the networks if the PN device name is similair to the configured device name
	                FOR #ti_LcPNDeviceNumber := 0 TO (#ti_NrOfDevices - 1) DO

	                    #iqUDT_PND.PNDeviceNumber := #ti_LcPNDeviceNumber;

	                    // set device found when a match is found for the device name in the PN network
	                    IF (#is_PNDeviceName = "DB_ProfinetDiagnostic".ProfinetNetworks[#iqUDT_PND.PNNetworknumber].DeviceStatus[#iqUDT_PND.PNDeviceNumber].DeviceState.PNDeviceName
	                        AND #is_PNDeviceName <> '')
	                    THEN

	                        #iqUDT_PND.PNDeviceFound := TRUE;
	                        EXIT;

	                    END_IF;
	                END_FOR;

	                // exit loop when device name is matching
	                IF #iqUDT_PND.PNDeviceFound
	                THEN

	                    EXIT;

	                END_IF;
	            END_FOR;
	        END_IF;
	    END_IF;

	END_REGION
END_FUNCTION

TYPE "UDT_PECUpdateConfiguration"
TITLE = UDT_PECConfiguration
VERSION : 0.1
//User-defined structure of PEC parameters.
   STRUCT
      Distance : DInt;   // Distance between photo eye and the end of conveyor [mm]
      JamDisplacementLimit : Int;   // Limit displacement with PEC blocked o detect jam [cm]
      TimeOnDelay : UDInt;   // Photo eye time on delay [ms]
      TimeOffDelay : UDInt;   // Photo eye time off delay [ms]
      ParcelLengthFilter : Bool := TRUE;   // Parcel length filter
      ResetWithPECBlocked { ExternalAccessible := 'False'; ExternalVisible := 'False'; ExternalWritable := 'False'} : Bool;   // When 'True' Allow reset system after jam with PEC blocked
      SearchWindowFwd : Int;   // Search window in forward direction [cm]
      SearchWindowRvs : Int;   // Search window in reverse direction [cm]
      GINRangeStart : Int;   // GIN range start value
      GINRangeEnd : Int;   // GIN range end value
      NrOfTeachParcels : Int;   // Number of parcels to teach
      DefaultGIN : Int := 1;   // Default GIN record
      MaxLost : Int;   // Maximum number of lost parcels in a row
      GenerationPoint { ExternalAccessible := 'False'; ExternalVisible := 'False'; ExternalWritable := 'False'} : Bool;   // Generation point
      NegativeGINDelete { ExternalAccessible := 'False'; ExternalVisible := 'False'; ExternalWritable := 'False'} : Bool;   // True when negative GIN has to be deleted
      ParcelLengthMeasurement { ExternalAccessible := 'False'; ExternalVisible := 'False'; ExternalWritable := 'False'} : Bool;   // Parcel length measurement
      GapLengthMeasurement { ExternalAccessible := 'False'; ExternalVisible := 'False'; ExternalWritable := 'False'} : Bool;   // Gap length measurement
   END_STRUCT;

END_TYPE

FUNCTION_BLOCK "FB_Conveyor"
TITLE = FB_Conveyor_BiDirectional
{ S7_Optimized_Access := 'TRUE' }
AUTHOR : MHSE
FAMILY : Equimpent
VERSION : 3.0
// ATTRIBUTES
// AUTO_NUMBER = True
// BLOCK_NUMBER = 207
// END_ATTRIBUTES
//Function block to control the bi-directional conveyor.
   VAR_INPUT
      iUDT_ConveyorConfiguration { ExternalAccessible := 'False'; ExternalVisible := 'False'; ExternalWritable := 'False'} : "UDT_ConveyorConfiguration";   //           Conveyor configuration structure
      idi_PECEoSDistance { ExternalAccessible := 'False'; ExternalVisible := 'False'; ExternalWritable := 'False'} : DInt;   //           Distance between photo eye and the end of conveyor [mm] in forward direction
      idi_PECBoSDistance { ExternalAccessible := 'False'; ExternalVisible := 'False'; ExternalWritable := 'False'} : DInt;   //           Distance between photo eye and the end of conveyor [mm] in reverse direction
      ii_ExternalSpeed { ExternalAccessible := 'False'; ExternalVisible := 'False'; ExternalWritable := 'False'} : Int;   //           External speed [mm/s]
      ix_SafetyOk { ExternalAccessible := 'False'; ExternalVisible := 'False'; ExternalWritable := 'False'} : Bool;   //           TRUE when safety is ok
      ix_24vOk { ExternalAccessible := 'False'; ExternalVisible := 'False'; ExternalWritable := 'False'} : Bool;   //           TRUE when 24VDC is healthy
      ix_400vOk { ExternalAccessible := 'False'; ExternalVisible := 'False'; ExternalWritable := 'False'} : Bool;   //           TRUE when 400VAC is healthy
      ix_HardwareOk { ExternalAccessible := 'False'; ExternalVisible := 'False'; ExternalWritable := 'False'} : Bool;   //           TRUE when  hardware is Ok
      ix_PECEoS { ExternalAccessible := 'False'; ExternalVisible := 'False'; ExternalWritable := 'False'} : Bool := TRUE;   //           TRUE when the end of section photoeye in forward direction is not blocked
      ix_PECBoS { ExternalAccessible := 'False'; ExternalVisible := 'False'; ExternalWritable := 'False'} : Bool := TRUE;   //           TRUE when the end of section photoeye in reverse direction is not blocked
      ix_ReverseDirection { ExternalAccessible := 'False'; ExternalVisible := 'False'; ExternalWritable := 'False'} : Bool;   //           FALSE when to run in forward direction and True to run in Reverse direction
      ix_ExternalRequestDieBack { ExternalAccessible := 'False'; ExternalVisible := 'False'; ExternalWritable := 'False'} : Bool;   //           External input to request die back
      ix_ExternalRequestHold { ExternalAccessible := 'False'; ExternalVisible := 'False'; ExternalWritable := 'False'} : Bool;   //           External input to request conveyor hold
      ix_ResetEnergySave { ExternalAccessible := 'False'; ExternalVisible := 'False'; ExternalWritable := 'False'} : Bool;   //           Reset energy save mode timer
   END_VAR

   VAR_OUTPUT
      qUDT_HMIStatus { ExternalAccessible := 'False'; ExternalVisible := 'False'; ExternalWritable := 'False'} : "UDT_ConveyorStatus";   //           HMI status structure
      qUDT_Status { ExternalAccessible := 'False'; ExternalVisible := 'False'; ExternalWritable := 'False'} : "UDT_CommonStatus";   //           Common status structure
   END_VAR

   VAR_IN_OUT
      iqUDT_EquipmentControl : "UDT_EquipmentControl";   //           Equipment control structure
      iqUDT_ConveyorCommand : "UDT_ConveyorCommand";   //           Conveyor command stucture
      iqUDT_ConveyorInterface : "UDT_ConveyorInterface";   //           Interface structure
      iqUDT_HandShakeUp : "UDT_ConveyorHandshake";   //           Upstream handshake structure in forward direction
      iqUDT_HandShake : "UDT_ConveyorHandshake";   //           Handshake structure in forward direction
      iqUDT_Statistics : "UDT_ConveyorStatistics";   //           Statistics structure
   END_VAR

